// ---- FBs_SlaveControllers/FB_SlaveCtrlMasterSlave.TcPOU
// Brief: Slave Arm MasterSlave controller
FUNCTION_BLOCK PUBLIC FB_SlaveCtrlMasterSlave EXTENDS FB_SlaveArmCtrlBase
VAR_INPUT
END_VAR
VAR_OUTPUT
END_VAR
VAR
	// pose track control kp
	m_posTrackKp :REAL := 0;
	m_oriTrackKp :REAL := 100;
	
	// minimum distance between instrument tip and remote center
	m_minInstruRCDis:LREAL := 0.05;
	
	// master-slave motion scale
	m_MSMotionScale :LREAL;
		
	// gripper match angle threshold
	m_gripperMatchAngThres :LREAL := 2*g_deg2Rad;
	
	// control error thershold from joint limit back to free space
	m_jntLimitOriErr :LREAL :=g_deg2Rad * 5;
	
	// master-slave error thershold to halt control 
	m_safetyOriErr :LREAL :=g_deg2Rad * 150;
	
	// filter cut-off frequency for master-slave control
	m_macroCmdJntPosLpfCutoffFreq : LREAL :=5;
	m_microCmdJntPosLpfCutoffFreq : LREAL :=15;
	
	// last command joint position
	m_lastCmdJntPos :Vec8d;
	
	// simulated DH joint position
	m_simDHJntPos : Vec6d;
	
	// simulated slave twist of DH joint
	m_simDHJointVel :Vec6d;
		
	// enter master-slave control for the first time
	m_firstIn :BOOL := TRUE;
	
	// flag if reach joint limit
	m_reachMacroJntLimit :BOOL;
	m_reachWristJntLimit :BOOL;
	m_jntLimitFlag :Vec6b;
	
	// master/slave origin pose when first enter master-slave control
	m_masterOriginPose : ST_Frame;
	m_slaveOriginPose : ST_Frame;
	
	// orientation deviation(in master coordinate) between master and slave when first enter control
	m_MSOriDeviation : Mat3d;
	
	// command joint position filter
	m_cmdJntPosLpf:ARRAY[1..8] OF FB_LowPassFilter;
	
	// commmand yaw angle and velocity
	m_cmdYawAngle :LREAL;
	m_cmdYawVel :LREAL;
	
	// comand yaw angle and velocity filter
	m_cmdYawAngLpf : FB_LowPassFilter;
	m_cmdYawVelLpf : FB_LowPassFilter;
	
	// master pose/velocity in monitor coordinate
	m_masterPose :ST_Frame;
	m_masterTwist : Vec6d;
	
	// master grip angle
	m_masterGripAngle : LREAL;
	
	// slave command/current pose in endoscope coordinate
	m_slaveCmdPoseInScope :ST_Frame;
	m_slavePoseInScope : ST_Frame;
	
	// slave command/current pose in cart
	m_slaveCmdPoseInCart :ST_Frame;
	m_slavePoseInCart : ST_Frame;
	
	// instrument controller
	m_basicInstruController : FB_BasicInstruControl;
	m_usKnifeController : FB_UltrosonicKnifeControl;
	
	// slave command grip angle and grip force level
	m_slaveCmdGripAngle :LREAL;
	m_slaveCmdGripForceLevel:LREAL;
	
	// slave pose error
	m_slavePosErr :Vec3d;
	m_slaveRotErr :Mat3d;
	m_errAngle : LREAL;
	m_errAxisLocal, m_errAxis :Vec3d;
	m_masterSlavePoseError :Vec6d;
	
	// master velocity in slave coordinate
	m_masterFFVel, m_masterFFWVel :Vec3d;
	
	// velocity for slave to track master motion
	m_slaveCmdVel, m_slaveCmdWVel : Vec3d;
	
	// flag to start gripper control
	m_gripperCtrlFlag :BOOL;
	
	// instrument tyep
	m_instruType : E_InstrumentType;
	
	//################# variable to interpolate master pose ##############
	m_firstInterpolate :BOOL :=TRUE;
	m_lastMasterPose : ST_Frame;
	m_lastMasterGripAngle :LREAL;
	m_masterInterpolateCycle :INT := 4;
	m_curInterpolateCylce :INT := 1;
	m_masterPosInterStep :Vec3d;
	m_masterOriInterStep :Mat3d;
	m_masterGripAngleInterStep :LREAL;
	m_interplotedMasterPose :ST_Frame;
	m_interplotedMasterGripAngle :LREAL;
	
	// code execute time measure
	m_codeTime : Profiler;
	
		m_jnt3Limit :LREAL;
		m_jnt3UB, m_jnt3LB :LREAL;
END_VAR

METHOD PROTECTED calcCmdJntPos : BOOL
VAR_IN_OUT CONSTANT
	i_endoscopePose : ST_Frame;
	i_masterStatus :ST_MasterStatus;
	i_setupStatus: ST_SetupStatus;
	i_slaveArm :FB_SlaveArm;
END_VAR

VAR 
	i,j : INT;
	tmpMat3d : Mat3d;
	masterMotionRange : Vec3d;
	
	masterVelInScope, masterWVelInScope :Vec3d;
	masterVelInCart, masterWVelInCart :Vec3d;

	cmdVelScale :LREAL;
	invJaco :Mat6d;
	armJntJaco,armJntJacoInv, wristJntJaco :Mat3d;
	velByWristJnt,velByArmJnt : Vec3d;
	armDHJntVel, wristDHJntVel :Vec3d;
	tmpFrame : ST_Frame;
	jnt3Limit :LREAL;
	jntDynaUB, jntDynaLB :LREAL;
END_VAR
m_codeTime(START:=TRUE, RESET:=TRUE);

IF isFinished THEN
	RETURN;
END_IF

// decide matched master arm index
FOR i:=1 TO g_mArmNum DO 
	IF i_masterStatus.m_teleSlaveArmIdx[i] = i_slaveArm.armIdx THEN
		masterPoseInterploate(i_masterStatus.m_curArmPose[i],i_masterStatus.m_gripAngle[i]);
		m_masterPose := m_interplotedMasterPose;
		m_masterGripAngle := m_interplotedMasterGripAngle;
		m_masterTwist := i_masterStatus.m_curArmTwist[i];
	END_IF
END_FOR

// compute slave pose in endoscope coordinate
m_slavePoseInCart := transform(i_setupStatus.m_curEndPose[i_slaveArm.armIdx], i_slaveArm.simCartPose);
tmpFrame :=invFrame(i_endoscopePose);
m_slavePoseInScope := transform(tmpFrame, m_slavePoseInCart);

// handle for the first time in
IF TRUE = m_firstIn THEN
	m_firstIn := FALSE;
	m_masterOriginPose :=m_masterPose;
	m_slaveOriginPose := m_slavePoseInScope;
	matTranspose(m_masterOriginPose.m_rot, tmpMat3d);
	matMultiply(tmpMat3d, m_slavePoseInScope.m_rot,m_MSOriDeviation);
	m_lastMasterGripAngle := m_masterGripAngle;
	
	// only update motion scale while entering teleControl 
	m_MSMotionScale := 1.0/ MAX(1,  i_masterStatus.m_motionScale);
END_IF

// compute master twist in slave arm coordinate
FOR i:=1 TO 3 DO
	masterVelInScope[i] := m_masterTwist[i]*m_MSMotionScale;
	masterWVelInScope[i] := m_masterTwist[i+3];
END_FOR
matMultiVec(i_endoScopePose.m_rot, masterVelInScope, masterVelInCart);
matMultiVec(i_endoScopePose.m_rot, masterWVelInScope, masterWVelInCart);
matTranspose(i_setupStatus.m_curEndPose[i_slaveArm.armIdx].m_rot, tmpMat3d);
matMultiVec(tmpMat3d,masterVelInCart, m_masterFFVel);
matMultiVec(tmpMat3d,masterWVelInCart, m_masterFFWVel);

// compute slave command pose in scope
vecSub(m_masterPose.m_pos, m_masterOriginPose.m_pos, masterMotionRange);
vecSelfMultiNum(masterMotionRange, m_MSMotionScale);
vecAdd(m_slaveOriginPose.m_pos, masterMotionRange, m_slaveCmdPoseInScope.m_pos);
matMultiply(m_masterPose.m_rot, m_MSOriDeviation, m_slaveCmdPoseInScope.m_rot);

// compute slave command pose in slave arm coordinate
m_slaveCmdPoseInCart := transform(i_endoScopePose, m_slaveCmdPoseInScope);
tmpFrame := invFrame(i_setupStatus.m_curEndPose[i_slaveArm.armIdx]);
m_cmdCartPose := transform(tmpFrame, m_slaveCmdPoseInCart);

// compute pose error
vecSub(m_cmdCartPose.m_pos, i_slaveArm.simCartPose.m_pos, m_slavePosErr);
matTranspose(i_slaveArm.simCartPose.m_rot, tmpMat3d);
matMultiply(tmpMat3d, m_cmdCartPose.m_rot, m_slaveRotErr);
rot2AngAxis(m_slaveRotErr, angle=>m_errAngle, axis=>m_errAxisLocal);
matMultiVec(i_slaveArm.simCartPose.m_rot, m_errAxisLocal, m_errAxis);

// calculate pose error in endoscope
calcMSErrInScope(i_endoscopePose, i_setupStatus.m_curEndPose[i_slaveArm.armIdx], i_slaveArm);

//safety check
IF ABS(m_errAngle)>m_safetyOriErr THEN
	m_isFinished := TRUE;
	RETURN;
END_IF

// pose track control
vecMultiNum(m_slavePosErr, m_posTrackKp, m_slaveCmdVel);
vecMultiNum(m_errAxis, m_errAngle*m_oriTrackKp, m_slaveCmdWVel);
// final command twist
FOR i:=1 TO 3 DO 
	m_cmdCartTwist[i] := m_slaveCmdVel[i] + m_masterFFVel[i];
	m_cmdCartTwist[i+3] := m_slaveCmdWVel[i] + m_masterFFWVel[i];
END_FOR

// compute command velocity for DH joints
invJaco := i_slaveArm.simJacoInv;
matMultiVec(invJaco, m_cmdCartTwist, m_simDHJointVel);

// limit instrument wrist dofs
limitInstruDofs(i_slaveArm, m_simDHJointVel);

// limit instrument wrist joint velocity
wristLimitSolve(i_slaveArm);

// limit DH joints velocity 
FOR i:=4 TO 6 DO 
	m_simDHJointVel[i] := LIMIT(-GVL_SlaveMotorParameters.g_maxJntVel[i], m_simDHJointVel[i], GVL_SlaveMotorParameters.g_maxJntVel[i]);
END_FOR

// modify arm joints velocity to compensate wrist joint motion
FOR i:=1 TO 3 DO
	FOR j:=1 TO 3 DO
		armJntJaco[i,j]:=i_slaveArm.simJaco[i,j];
		wristJntJaco[i,j]:=i_slaveArm.simJaco[i,j+3];
	END_FOR
	armDHJntVel[i]:=m_simDHJointVel[i];
	wristDHJntVel[i]:=m_simDHJointVel[i+3];
	m_slaveCmdVel[i] := m_cmdCartTwist[i];
END_FOR
invMat3(armJntJaco, armJntJacoInv);
matMultiVec(wristJntJaco, wristDHJntVel, velByWristJnt);
vecSub(m_slaveCmdVel, velByWristJnt, velByArmJnt);
matMultiVec(armJntJacoInv, velByArmJnt, armDHJntVel);

// limit arm joint position
m_reachMacroJntLimit:=false;
FOR i:=1 TO 3 DO
	jntDynaLB := MIN( 0, (GVL_SlaveMotorParameters.g_minDHJntPos[i] - i_slaveArm.simDHJntPos[i])/g_slaveArmCtrlCycleTime);
	IF i=3 THEN
		jnt3Limit := i_slaveArm.instrument.kinematicParameters.m_rodLength+i_slaveArm.instrument.kinematicParameters.m_headLength
											+ i_slaveArm.instrument.kinematicParameters.m_fingerLength - GVL_SlaveArmKinematic.g_minInstruRCDis;
		jntDynaUB := MAX( 0, (jnt3Limit - i_slaveArm.simDHJntPos[i])/g_slaveArmCtrlCycleTime);
		m_jnt3Limit := jnt3Limit;
		m_jnt3UB :=jntDynaUB;
		m_jnt3LB := jntDynaLB;
	ELSE
		jntDynaUB := MAX( 0, (GVL_SlaveMotorParameters.g_maxDHJntPos[i] - i_slaveArm.simDHJntPos[i])/g_slaveArmCtrlCycleTime);
	END_IF
	
	IF m_simDHJointVel[i] >= jntDynaUB OR m_simDHJointVel[i]<= jntDynaLB THEN
		armDHJntVel[i]:=LIMIT(jntDynaLB, m_simDHJointVel[i], jntDynaUB);
		m_reachMacroJntLimit:=TRUE;
	END_IF
END_FOR

// limit DH joints velocity 
FOR i:=1 TO 3 DO
	m_simDHJointVel[i]:=armDHJntVel[i];
	m_simDHJointVel[i+3]:=wristDHJntVel[i];
END_FOR
cmdVelScale := 1;
FOR i:=1 TO g_cartDofs DO 
	cmdVelScale:=MAX(cmdVelScale, ABS(m_simDHJointVel[i]/GVL_SlaveMotorParameters.g_maxJntVel[i]));
END_FOR
vecSelfMultiNum(m_simDHJointVel, 1.0/cmdVelScale);

// integrate command DH joint position
FOR i:=1 TO 6 DO
	m_simDHJntPos[i] := i_slaveArm.simDHJntPos[i] + m_simDHJointVel[i]*g_slaveArmCtrlCycleTime;
END_FOR

// gripper angle/force control
gripperControl(i_slaveArm);

// calculate target motor joint position/velocity from DH joint position
i_slaveArm.instrument.instruIK(m_simDHJntPos,m_slaveCmdGripAngle, o_jntPos=>m_simJntPos);

// filt command joint position
FOR i:=1 TO g_sJntNum DO 
	m_cmdJntPos[i] := m_cmdJntPosLpf[i].run(m_simJntPos[i]);
END_FOR

// compute command joint velocity
vecSub(m_cmdJntPos, m_lastCmdJntPos, m_cmdJntVel);
vecSelfMultiNum(m_cmdJntVel, g_slaveArmCtrlFreq);
m_lastCmdJntPos:=m_cmdJntPos;

m_codeTime(START:=FALSE);
END_METHOD

// override this function in each exact controller
METHOD PROTECTED calcCmdJntTrq : BOOL
VAR_IN_OUT CONSTANT
	i_endoscopePose : ST_Frame;
	i_masterStatus :ST_MasterStatus;
	i_setupStatus: ST_SetupStatus;
	i_slaveArm :FB_SlaveArm;
END_VAR
VAR
	i :INT ;
	instruCmdGripAngle, instruCmdGripForceLevel :LREAL;
	instruCmdJntPos, instruCmdJntVel : Vec5d;	
	instruJntCtrlTrq :Vec5d;
END_VAR
IF isFinished THEN
	RETURN;
END_IF

// set joint torque to zero in default
m_cmdJntTrq := g_zeroVec8d;

// instrument joint control
FOR i:=1 TO 5 DO 
	instruCmdJntPos[i]:=m_cmdJntPos[i+3];
	instruCmdJntVel[i]:=m_cmdJntVel[i+3];
END_FOR
m_cmdYawAngle := m_cmdYawAngLpf.run(m_simDHJntPos[6]);
m_cmdYawVel := m_cmdYawVelLpf.run(m_simDHJointVel[6]);

IF i_slaveArm.instrument.instruType = InstruType_UltrasoundKnifeS OR i_slaveArm.instrument.instruType = InstruType_UltrasoundKnifeU THEN
	m_usKnifeController.run(instruCmdJntPos,instruCmdJntVel, m_slaveCmdGripForceLevel, i_slaveArm, o_cmdJntTrq=>instruJntCtrlTrq);
ELSE
	m_basicInstruController.run(instruCmdJntPos,instruCmdJntVel, m_cmdYawAngle, m_cmdYawVel, m_slaveCmdGripForceLevel, i_slaveArm, o_cmdJntTrq=>instruJntCtrlTrq);
END_IF

FOR i:=1 TO 5 DO
	m_cmdJntTrq[i+3]:=instruJntCtrlTrq[i];
END_FOR
END_METHOD

METHOD calcMSErrInScope : BOOL
VAR_IN_OUT CONSTANT
	i_endoscopePose : ST_Frame;
	i_setupPose :ST_Frame;
	i_slaveArm :FB_SlaveArm;
END_VAR
VAR
	posErrInCart,oriErrInCart :Vec3d;
	invRot :Mat3d;
	posErrInScope,oriErrInScope :Vec3d;
	i:INT;
END_VAR
m_masterSlavePoseError := g_zeroVec6d;

// pose error caused by joints limits
IF m_reachMacroJntLimit OR m_reachWristJntLimit THEN
	// pose error in cart coordinate
	matMultiVec(i_setupPose.m_rot, m_slavePosErr, posErrInCart);
	matMultiVec(i_setupPose.m_rot, m_errAxis, oriErrInCart);
	vecSelfMultiNum(oriErrInCart, m_errAngle);
	
	// pose err in endoscope coordinate
	matTranspose(i_endoscopePose.m_rot, invRot);
	matMultiVec(invRot, posErrInCart, posErrInScope);
	matMultiVec(invRot, oriErrInCart, oriErrInScope);
	
	FOR i:=1 TO 3 DO 
		m_masterSlavePoseError[i]:=posErrInScope[i];
		m_masterSlavePoseError[i+3]:=oriErrInScope[i];
	END_FOR

END_IF
END_METHOD

METHOD gripperControl : BOOL
VAR_IN_OUT CONSTANT
	i_slaveArm :FB_SlaveArm;
END_VAR

VAR
	matchedSlaveGripAngle:LREAL;
	matchedSlaveGripForce:LREAL;
	masterGripVelThres :LREAL := 5.0 *g_deg2Rad;
END_VAR
// compute matched slave grip angle and force
i_slaveArm.instrument.gripAngleMap(m_masterGripAngle,o_instruGripAngle=>matchedSlaveGripAngle, o_instruGripForceLevel=>matchedSlaveGripForce);

IF m_gripperCtrlFlag THEN
	m_slaveCmdGripAngle := matchedSlaveGripAngle;
	m_slaveCmdGripForceLevel := matchedSlaveGripForce;
	RETURN;
ELSE
	//m_gripperCtrlFlag := (ABS(m_masterGripAngleVel) >masterGripVelThres) AND  (m_masterGripAngleVel * (matchedSlaveGripAngle-i_slaveArm.curGripAngle)>0);
	m_gripperCtrlFlag := ABS(matchedSlaveGripAngle-i_slaveArm.curGripAngle)<m_gripperMatchAngThres OR 
	     (matchedSlaveGripAngle>=i_SlaveArm.instrument.kinematicParameters.m_maxGripAngle - m_gripperMatchAngThres AND i_slaveArm.curGripAngle>=matchedSlaveGripAngle) OR 
		(matchedSlaveGripAngle<=i_SlaveArm.instrument.kinematicParameters.m_minGripAngle + m_gripperMatchAngThres AND i_slaveArm.curGripAngle<=matchedSlaveGripAngle);
END_IF
END_METHOD

METHOD PUBLIC init : BOOL
VAR_IN_OUT CONSTANT
	i_slaveArm	:FB_SlaveArm;
END_VAR
VAR_IN_OUT 
	r_slaveArmCtrlCmd :ST_SlaveArmCtrlCmds;
END_VAR
VAR 
	i :INT ;
END_VAR
SUPER^.Init(i_slaveArm,r_slaveArmCtrlCmd);
m_simJntPos :=m_cmdJntPos;
m_lastCmdJntPos :=m_cmdJntPos;
m_jntOPMode[1] := DriverOPMode_PosTrq;
m_jntOPMode[2] := DriverOPMode_PosTrq;
m_jntOPMode[3] := DriverOPMode_PosTrq;
m_jntOPMode[4] := DriverOPMode_Trq;
m_jntOPMode[5] := DriverOPMode_Trq;
m_jntOPMode[6] := DriverOPMode_Trq;
m_jntOPMode[7] := DriverOPMode_Trq;
m_jntOPMode[8] := DriverOPMode_Trq;
m_firstIn :=TRUE;
m_gripperCtrlFlag :=FALSE;

// init gripper angle
m_slaveCmdGripAngle := i_slaveArm.curGripAngle;
m_slaveCmdGripForceLevel:=0;

// init filter
FOR i:=1 TO 3 DO
	m_cmdJntPosLpf[i].init(1, m_macroCmdJntPosLpfCutoffFreq, g_slaveArmCtrlFreq);
END_FOR
FOR i:=4 TO g_sJntNum DO
	m_cmdJntPosLpf[i].init(1, m_microCmdJntPosLpfCutoffFreq, g_slaveArmCtrlFreq);
END_FOR
m_cmdYawAngLpf.init(1, m_microCmdJntPosLpfCutoffFreq, g_slaveArmCtrlFreq);
m_cmdYawVelLpf.init(1, m_microCmdJntPosLpfCutoffFreq, g_slaveArmCtrlFreq);

// init controller
m_basicInstruController.init(i_slaveArm);
m_usKnifeController.init(i_slaveArm);
m_instruType := i_slaveArm.instrument.instruType;

// init interpolation data
m_firstInterpolate :=TRUE;
m_curInterpolateCylce := 1;

// update commands to arm
copyCmds(r_slaveArmCtrlCmd);
END_METHOD

PROPERTY InstruBacklash : Vec5d
GET
IF m_instruType = InstruType_UltrasoundKnifeS OR m_instruType = InstruType_UltrasoundKnifeU THEN
	instruBacklash := g_zeroVec5d;
ELSE
	instruBacklash := m_basicInstruController.m_jntBacklash;
END_IF
END_GET
END_PROPERTY

// limit specific joint dofs based on instrument types
METHOD PRIVATE limitInstruDofs : BOOL
VAR_IN_OUT CONSTANT
	i_slaveArm :FB_SlaveArm;
END_VAR

VAR_IN_OUT
	r_simDHJointVel :Vec6d;
END_VAR
IF i_slaveArm.instrument.instruType = InstruType_UltrasoundKnifeS OR i_slaveArm.instrument.instruType = InstruType_UltrasoundKnifeU THEN
	r_simDHJointVel[5] :=0;
	r_simDHJointVel[6] :=0;
END_IF
END_METHOD

// every some cycles the data from master robots would be miss, so add this interpolation
METHOD masterPoseInterploate : BOOL
VAR_INPUT
	i_masterPose :ST_FRAME;
	i_masterGripAngle :LREAL;
END_VAR

VAR
	rotT :Mat3d;
	rotErr:Mat3d;
	errAngle:LREAL;
	errAxisLocal :Vec3d;
	tmpMat :Mat3d;
END_VAR
IF m_firstInterpolate THEN
	m_firstInterpolate :=FALSE;
	m_lastMasterGripAngle :=i_masterGripAngle;
	m_lastMasterPose := i_masterPose;
	m_masterPosInterStep :=g_zeroVec3d;
	m_masterOriInterStep :=g_eye3d;
	m_masterGripAngleInterStep :=0.0;
	m_interplotedMasterPose := i_masterPose;
	m_interplotedMasterGripAngle := i_masterGripAngle;
END_IF


// update next interpolation
IF m_curInterpolateCylce > m_masterInterpolateCycle THEN
	vecSub(i_masterPose.m_pos, m_lastMasterPose.m_pos, m_masterPosInterStep);
	vecSelfMultiNum( m_masterPosInterStep, 1.0/INT_TO_LREAL(m_masterInterpolateCycle));
	
	matTranspose(m_lastMasterPose.m_rot, rotT);
	matMultiply(rotT, i_masterPose.m_rot, rotErr);
	rot2AngAxis(rotErr, angle=>errAngle, axis=>errAxisLocal);
	m_masterOriInterStep := angAxis2Rot(errAngle/INT_TO_LREAL(m_masterInterpolateCycle), errAxisLocal);
	
	m_masterGripAngleInterStep := (i_masterGripAngle- m_lastMasterGripAngle)/INT_TO_LREAL(m_masterInterpolateCycle);
	
	m_curInterpolateCylce :=1;
	m_lastMasterPose:= i_masterPose;
	m_lastMasterGripAngle := i_masterGripAngle;
END_IF

// control points
IF m_curInterpolateCylce = m_masterInterpolateCycle THEN
	m_interplotedMasterGripAngle := m_lastMasterGripAngle;
	m_interplotedMasterPose := m_lastMasterPose;
// interpolation
ELSE
	m_interplotedMasterGripAngle := m_interplotedMasterGripAngle + m_masterGripAngleInterStep;
	vecSelfAdd(m_interplotedMasterPose.m_pos, m_masterPosInterStep);
	tmpMat := m_interplotedMasterPose.m_rot;
	matMultiply(tmpMat, m_masterOriInterStep, m_interplotedMasterPose.m_rot);
END_IF

m_curInterpolateCylce:= m_curInterpolateCylce+1;
END_METHOD

PROPERTY masterSlavePoseErr : REFERENCE to Vec6d
GET
masterSlavePoseErr REF= m_masterSlavePoseError;
END_GET
END_PROPERTY

// calculate optimized wrist joint velocity when joint limit is violated
METHOD wristLimitSolve : BOOL
VAR_IN_OUT CONSTANT
	i_slaveArm :FB_SlaveArm;
END_VAR

VAR
	i,j:INT;
	jntDynaUB, jntDynaLB :LREAL;
	
	dsrWVel:Vec3d;
	wristJntVel :Vec3d;
	wristJaco:Mat3d;
	
	optJntVel:Vec2d;
	partJaco :Mat32;
	partJacoT :Mat23;
	JtJ,JtJInv :Mat2d;
	partJacoPInv:Mat23;
	
	partJacoPinv2 :Vec3d;
	jacoNorm :LREAL;
	
	wVelLocal,wVelWrd:Vec3d;
	matT:Mat3d;
END_VAR
m_reachWristJntLimit := FALSE;

// desire angular velocity from wrist joint
FOR i:=1 TO 3 DO
	wristJntVel[i] := m_simDHJointVel[i+3];
	FOR j:=1 TO 3 DO
		wristJaco[i,j]:= i_slaveArm.simJaco[i+3, j+3];
	END_FOR 
END_FOR
matMultiVec(wristJaco, wristJntVel, dsrWVel);

// check which joint reaches limit
FOR i:=4 TO 6 DO
	m_jntLimitFlag[i] := FALSE;
	jntDynaUB := MAX( 0, (i_slaveArm.instrument.kinematicParameters.m_wristMaxDHJntPos[i-3] - i_slaveArm.simDHJntPos[i])/g_slaveArmCtrlCycleTime);
	jntDynaLB := MIN( 0, (i_slaveArm.instrument.kinematicParameters.m_wristMinDHJntPos[i-3] - i_slaveArm.simDHJntPos[i])/g_slaveArmCtrlCycleTime);
	IF m_simDHJointVel[i] >= jntDynaUB OR m_simDHJointVel[i]<=jntDynaLB THEN
		m_simDHJointVel[i]:=LIMIT(jntDynaLB, m_simDHJointVel[i], jntDynaUB);
		m_jntLimitFlag[i]:=TRUE;
		m_reachWristJntLimit := TRUE;
	END_IF
END_FOR

// no limit violated
IF NOT( m_jntLimitFlag[4]) AND NOT(m_jntLimitFlag[5]) AND NOT(m_jntLimitFlag[6]) THEN
	RETURN;
END_IF; 

// all joint reach limit
IF m_jntLimitFlag[4] AND m_jntLimitFlag[5] AND m_jntLimitFlag[6] THEN
	RETURN;
END_IF;

// joint 4 reach limit
IF m_jntLimitFlag[4] AND NOT(m_jntLimitFlag[5]) AND NOT(m_jntLimitFlag[6]) THEN
	// colume 2/3
	partJaco[1,1]:= wristJaco[1,2];
	partJaco[2,1]:= wristJaco[2,2];
	partJaco[3,1]:= wristJaco[3,2];
	
	partJaco[1,2]:= wristJaco[1,3];
	partJaco[2,2]:= wristJaco[2,3];
	partJaco[3,2]:= wristJaco[3,3];
	
	// pinv partJaco
	matTranspose(partJaco, partJacoT);
	matMultiply(partJacoT, partJaco, JtJ);
	IF NOT(invMat2(JtJ, JtJInv)) THEN
		m_simDHJointVel[5] :=0;
		m_simDHJointVel[6] := 0;
		RETURN;
	END_IF
	matMultiply(JtJInv, partJacoT, partJacoPinv);
	
	// desire angular velocity exclusive limited joint motion
	dsrWVel[1] := dsrWVel[1] - wristJaco[1,1] * m_simDHJointVel[4];
	dsrWVel[2] := dsrWVel[2] - wristJaco[2,1] * m_simDHJointVel[4];
	dsrWVel[3] := dsrWVel[3] - wristJaco[3,1] * m_simDHJointVel[4];
	
	//NOTE: special handle for roll limit. avoiding joint5/6 motion caused by pitch limit
	matTranspose(i_slaveArm.simCartPose.m_rot, matT);
	matMultiVec(matT, dsrWVel, wVelLocal);
	wVelLocal[3]:=0;
	matMultiVec(i_slaveArm.simCartPose.m_rot, wVelLocal, dsrWVel);
	
	// solve
	matMultiVec(partJacoPinv, dsrWVel, optJntVel);
	m_simDHJointVel[5] :=optJntVel[1];
	m_simDHJointVel[6] := optJntVel[2];
END_IF

// joint 5 reach limit
IF m_jntLimitFlag[5] AND NOT(m_jntLimitFlag[4]) AND NOT(m_jntLimitFlag[6]) THEN
	// colume 1/3
	partJaco[1,1]:= wristJaco[1,1];
	partJaco[2,1]:= wristJaco[2,1];
	partJaco[3,1]:= wristJaco[3,1];
	
	partJaco[1,2]:= wristJaco[1,3];
	partJaco[2,2]:= wristJaco[2,3];
	partJaco[3,2]:= wristJaco[3,3];
	
	// pinv partJaco
	matTranspose(partJaco, partJacoT);
	matMultiply(partJacoT, partJaco, JtJ);
	IF NOT(invMat2(JtJ, JtJInv)) THEN
		m_simDHJointVel[4] :=0;
		m_simDHJointVel[6] := 0;
		RETURN;
	END_IF
	matMultiply(JtJInv, partJacoT, partJacoPinv);
		
	// desire angular velocity exclusive limited joint motion
	dsrWVel[1] := dsrWVel[1] - wristJaco[1,2] * m_simDHJointVel[5];
	dsrWVel[2] := dsrWVel[2] - wristJaco[2,2] * m_simDHJointVel[5];
	dsrWVel[3] := dsrWVel[3] - wristJaco[3,2] * m_simDHJointVel[5];
	
	//NOTE: special handle for pitch limit. avoiding joint4/6 motion caused by pitch limit
	matTranspose(i_slaveArm.simCartPose.m_rot, matT);
	matMultiVec(matT, dsrWVel, wVelLocal);
	wVelLocal[1]:=0;
	matMultiVec(i_slaveArm.simCartPose.m_rot, wVelLocal, dsrWVel);
	
	// solve
	matMultiVec(partJacoPinv, dsrWVel, optJntVel);
	m_simDHJointVel[4] :=optJntVel[1];
	m_simDHJointVel[6] := optJntVel[2];
END_IF

// joint 6 reach limit
IF m_jntLimitFlag[6] AND NOT(m_jntLimitFlag[4]) AND NOT(m_jntLimitFlag[5]) THEN
	// colume 1/2
	partJaco[1,1]:= wristJaco[1,1];
	partJaco[2,1]:= wristJaco[2,1];
	partJaco[3,1]:= wristJaco[3,1];
	
	partJaco[1,2]:= wristJaco[1,2];
	partJaco[2,2]:= wristJaco[2,2];
	partJaco[3,2]:= wristJaco[3,2];
	
	// pinv partJaco
	matTranspose(partJaco, partJacoT);
	matMultiply(partJacoT, partJaco, JtJ);
	IF NOT(invMat2(JtJ, JtJInv)) THEN
		m_simDHJointVel[4] :=0;
		m_simDHJointVel[5] := 0;
		RETURN;
	END_IF
	matMultiply(JtJInv, partJacoT, partJacoPinv);
		
	// desire angular velocity exclusive limited joint motion
	dsrWVel[1] := dsrWVel[1] - wristJaco[1,3] * m_simDHJointVel[6];
	dsrWVel[2] := dsrWVel[2] - wristJaco[2,3] * m_simDHJointVel[6];
	dsrWVel[3] := dsrWVel[3] - wristJaco[3,3] * m_simDHJointVel[6];
	
	// solve
	matMultiVec(partJacoPinv, dsrWVel, optJntVel);
	m_simDHJointVel[4] :=optJntVel[1];
	m_simDHJointVel[5] := optJntVel[2];
END_IF

// joint 4/5 reach limit
IF m_jntLimitFlag[4] AND m_jntLimitFlag[5] AND NOT(m_jntLimitFlag[6]) THEN
	// pinv partJaco of column 3
	partJacoPinv2[1] := wristJaco[1, 3];
	partJacoPinv2[2] := wristJaco[2, 3];
	partJacoPinv2[3] := wristJaco[3, 3];
	jacoNorm := norm(partJacoPinv2);
	vecSelfMultiNum(partJacoPinv2, 1.0/(jacoNorm*jacoNorm));
		
	// desire angular velocity exclusive limited joint motion
	dsrWVel[1] := dsrWVel[1] - wristJaco[1,1] * m_simDHJointVel[4] - wristJaco[1,2] * m_simDHJointVel[5];
	dsrWVel[2] := dsrWVel[2] - wristJaco[2,1] * m_simDHJointVel[4] - wristJaco[2,2] * m_simDHJointVel[5];
	dsrWVel[3] := dsrWVel[3] - wristJaco[3,1] * m_simDHJointVel[4] - wristJaco[3,2] * m_simDHJointVel[5];
	
	// solve
	m_simDHJointVel[6] := vecDot(partJacoPinv2, dsrWVel);
END_IF

// joint 4/6 reach limit
IF m_jntLimitFlag[4] AND m_jntLimitFlag[6] AND NOT(m_jntLimitFlag[5]) THEN
	// pinv partJaco of column 2
	partJacoPinv2[1] := wristJaco[1, 2];
	partJacoPinv2[2] := wristJaco[2, 2];
	partJacoPinv2[3] := wristJaco[3, 2];
	jacoNorm := norm(partJacoPinv2);
	vecSelfMultiNum(partJacoPinv2, 1.0/(jacoNorm*jacoNorm));
		
	// desire angular velocity exclusive limited joint motion
	dsrWVel[1] := dsrWVel[1] - wristJaco[1,1] * m_simDHJointVel[4] - wristJaco[1,3] * m_simDHJointVel[6];
	dsrWVel[2] := dsrWVel[2] - wristJaco[2,1] * m_simDHJointVel[4] - wristJaco[2,3] * m_simDHJointVel[6];
	dsrWVel[3] := dsrWVel[3] - wristJaco[3,1] * m_simDHJointVel[4] - wristJaco[3,3] * m_simDHJointVel[6];
	
	// solve
	m_simDHJointVel[5] := vecDot(partJacoPinv2, dsrWVel);
END_IF

// joint 5/6 reach limit
IF m_jntLimitFlag[5] AND m_jntLimitFlag[6] AND NOT(m_jntLimitFlag[4]) THEN
	// pinv partJaco of column 4
	partJacoPinv2[1] := wristJaco[1, 1];
	partJacoPinv2[2] := wristJaco[2, 1];
	partJacoPinv2[3] := wristJaco[3, 1];
	jacoNorm := norm(partJacoPinv2);
	vecSelfMultiNum(partJacoPinv2, 1.0/(jacoNorm*jacoNorm));
		
	// desire angular velocity exclusive limited joint motion
	dsrWVel[1] := dsrWVel[1] - wristJaco[1,2] * m_simDHJointVel[5] - wristJaco[1,3] * m_simDHJointVel[6];
	dsrWVel[2] := dsrWVel[2] - wristJaco[2,2] * m_simDHJointVel[5] - wristJaco[2,3] * m_simDHJointVel[6];
	dsrWVel[3] := dsrWVel[3] - wristJaco[3,2] * m_simDHJointVel[5] - wristJaco[3,3] * m_simDHJointVel[6];
	
	// solve
	m_simDHJointVel[4] := vecDot(partJacoPinv2, dsrWVel);
END_IF


// check which joint reaches limit
FOR i:=4 TO 6 DO
	jntDynaUB := MAX( 0, (i_slaveArm.instrument.kinematicParameters.m_wristMaxDHJntPos[i-3] - i_slaveArm.simDHJntPos[i])/g_slaveArmCtrlCycleTime);
	jntDynaLB := MIN( 0, (i_slaveArm.instrument.kinematicParameters.m_wristMinDHJntPos[i-3] - i_slaveArm.simDHJntPos[i])/g_slaveArmCtrlCycleTime);
	IF m_simDHJointVel[i] >= jntDynaUB OR m_simDHJointVel[i]<=jntDynaLB THEN
		m_simDHJointVel[i]:=LIMIT(jntDynaLB, m_simDHJointVel[i], jntDynaUB);
		m_jntLimitFlag[i]:=TRUE;
		m_reachWristJntLimit := TRUE;
	END_IF
END_FOR
END_METHOD

END_FUNCTION_BLOCK

// ---- Mains/SafetyCheck.TcPOU
PROGRAM SafetyCheck
VAR
	// slave robot information, including arm status and cartesian data
	m_slaveStatus AT %I* :ST_slaveStatus;
	
	// slave robot joint data
	m_slaveJointData AT %I* :ST_slaveJointData;
	
	// setup robot information
	m_setupStatus AT %I* :ST_SetupStatus;
	
	// setup robot joint data
	m_setupJointsData AT %I* :ST_SetupJointData;
	
	// master robot data, input from master controller box
	m_masterRobotData AT %I* : MSCommu_MasterStatus;
	
	// error check result
	m_safetyCheckData AT %Q* :ST_SafetyData;
	
	// Output cart status
	m_cartStatus AT%I* : ST_CartStatus;
	
	// cart joint data
	m_cartJointsData AT %I* :ST_CartJointData;
	
	//emergency stop and stop botton
	m_stopButton AT %I*: BOOL;
	m_emergencyStopButton AT %I*: BOOL;
	
	//warning tone
	m_warningTone AT %Q*:ARRAY [1..4] OF BOOL;
	
	m_initFlag:bool;
	
	m_SafetyCheck : Fb_SafetyCheck;
	m_checkVariable : ARRAY[1..g_maxNum] OF checkInputVariable;
	m_EtherCATCheck :ARRAY [1..g_maxNum,1..g_maxArmJoint] OF Fb_EtherCATCheck;
	m_errCode :ARRAY [1..3] OF UDINT;
	i , j: INT;
	
	//error robot data record
	m_dataRecord : Fb_dataRecord;
	
	// original position of remote center point when fisrt enter hold state
	m_dsrRcpPos :ARRAY[1..g_sArmNum] OF Vec3d;
	m_rcpPosErrCounts :ARRAY[1..g_sArmNum] OF INT := [4(0)];
	m_rcpPosErr :ARRAY[1..g_sArmNum] OF Vec3d;		// rcp position error
	m_curJntPosLast : ARRAY [1..g_maxArmNum] OF vec13di;  
	m_armErrCodeRefreshLast : ARRAY [1..4] OF UINT;
	
	m_armsRS:ARRAY [1..g_maxArmNum,1..30] OF RS;//复位优先双稳态器
	m_cartRS:ARRAY [1..30] OF RS;//复位优先双稳态器
	m_scopeArmNoReady : BOOL;
	m_joysticksTrigger : BOOL;
	// wait time before robot init  for ethercat to be statble 
	m_safetyCheckInitWaitTime : LREAL:=0;
	
	m_test : DINT;
END_VAR

// reset data
IF FALSE = m_initFlag  THEN
	FOR i:=1  TO g_sArmNum DO 
		m_safetyCheckData.m_slaveErrFlag[i]:=FALSE;
		m_safetyCheckData.m_setupErrFlag[i]:=FALSE;
		m_safetyCheckData.m_cartErrFlag:=FALSE;
	END_FOR
	m_initFlag:=TRUE;
END_IF

armSafetyCheckInputCast();

armSafetyCheckAllowed();

robotPromptMassageCast();

// wait communication to be stable
IF(m_safetyCheckInitWaitTime<g_robotSafetyCheckWaitTime) THEN
	m_safetyCheckInitWaitTime := m_safetyCheckInitWaitTime+g_setupArmCtrlCycleTime;
	RETURN;
END_IF


FOR i:=1  TO g_maxNum DO
	m_SafetyCheck.systemSafetyCheck(i,m_checkVariable,m_cartJointsData,m_setupJointsData,m_slaveJointData);
END_FOR


//error flag to control
readErrFlag();

//Fault code for UI
m_SafetyCheck.errCodeUpdating();

//The fault code is sent to the UI
GVL_interactUI.g_errIdType3:=m_SafetyCheck.o_ErrCode[3];
GVL_interactUI.g_errIdType2:=m_SafetyCheck.o_ErrCode[2];
GVL_interactUI.g_errIdType1:=m_SafetyCheck.o_ErrCode[1];
GVL_interactUI.g_popupErrorArm1 := m_SafetyCheck.m_armErrCodePopup[1];
GVL_interactUI.g_popupErrorArm2 := m_SafetyCheck.m_armErrCodePopup[2];
GVL_interactUI.g_popupErrorArm3 := m_SafetyCheck.m_armErrCodePopup[3];
GVL_interactUI.g_popupErrorArm4 := m_SafetyCheck.m_armErrCodePopup[4];
FOR i:=1  TO g_sArmNum DO
	IF m_SafetyCheck.m_armErrCodeRefresh[i] <> m_armErrCodeRefreshLast[i] THEN
		GVL_interactUI.g_popupRefresh[i] := 1;
	END_IF
	m_armErrCodeRefreshLast[i] := m_SafetyCheck.m_armErrCodeRefresh[i];
END_FOR

//clear fault
IF GVL_interactUI.g_uiFaultReset=1 OR m_masterRobotData.m_uiResetFault = 1 THEN
	m_SafetyCheck.errFlagReset();
	GVL_interactUI.g_uiFaultReset := 0;
END_IF

//robot record information
m_dataRecord.run(m_checkVariable , m_cartStatus , m_cartJointsData , m_setupStatus , m_slaveStatus , m_setupJointsData , m_slaveJointData );

//m_warningTone := warningTone();

METHOD armSafetyCheckAllowed : BOOL
VAR_INPUT
END_VAR
VAR
	i , j : INT; 
END_VAR
FOR i := 1 TO g_maxArmNum DO
	FOR j := 1 TO g_maxArmJoint DO
		IF j > 5 THEN
			//fault code 16#3003 
			m_SafetyCheck.checkPermit[i].m_linkEncErr[j] := m_checkVariable[i].m_slaveDriverInput[j-g_setupJntNum].m_statusWord<>0;
			//fault code 16#3002 
			m_SafetyCheck.checkPermit[i].m_currentIsNotUpdate[j] :=m_checkVariable[i].m_slaveDriverInput[j-g_setupJntNum].m_statusWord<>0 ;
			//fault code 16#2002
			m_SafetyCheck.checkPermit[i].m_armJntFollowErr[j] := m_checkVariable[i].m_slaveDriverInput[j-g_setupJntNum].m_statusWord = DriverStatusWord_OP ;
			//fault code 16#200B
			m_SafetyCheck.checkPermit[i].m_jntCurrentCtrlErr[j] := m_checkVariable[i].m_slaveDriverOutput[j-g_setupJntNum].m_opMode = DriverOPMode_Trq;
		ELSE
			//fault code 16#3003 
			m_SafetyCheck.checkPermit[i].m_linkEncErr[j] := m_checkVariable[i].m_setupDriverInput[j].m_statusWord<>0;
			//fault code 16#3002
			m_SafetyCheck.checkPermit[i].m_currentIsNotUpdate[j] := m_checkVariable[i].m_setupDriverInput[j].m_statusWord<>0 AND j > 2;
			//fault code 16#2002
			m_SafetyCheck.checkPermit[i].m_armJntFollowErr[j] := m_checkVariable[i].m_setupDriverInput[j].m_statusWord = DriverStatusWord_OP AND j > 2;
			//fault code 16#200B
			m_SafetyCheck.checkPermit[i].m_jntCurrentCtrlErr[j] := m_checkVariable[i].m_setupDriverOutput[j].m_opMode = DriverOPMode_Trq AND j > 2;
			
		END_IF
		//fault code 16#3002
		m_SafetyCheck.checkPermit[i].m_jntStatusErr[j] := TRUE;
		//fault code 16#3004
		m_SafetyCheck.checkPermit[i].m_driveErr[j] := TRUE;
		//fault code 16#3005
		m_SafetyCheck.checkPermit[i].m_armJntEncErr[j] := TRUE;
		//fault code 16#3006
		m_SafetyCheck.checkPermit[i].m_outOfLimit[j] := TRUE;
		//fault code 16#3008
		m_SafetyCheck.checkPermit[i].m_motPhieErr[j] := TRUE;
		//fault code 16#2003
		m_SafetyCheck.checkPermit[i].m_jntVelErr[j] := TRUE;
		//fault code 16#2004
		m_SafetyCheck.checkPermit[i].m_spacePoseErr[j] := m_slaveStatus.m_armState[i] = SlaveArmState_MasterSlave AND  norm(m_slaveStatus.m_masterSlavePoseError[i])<g_smallNum;
		//fault code 16#2005
		m_SafetyCheck.checkPermit[i].m_jntCurrentErr[j] := TRUE;
		//fault code 16#2007
		m_SafetyCheck.checkPermit[i].m_fixedPointErr := m_slaveStatus.m_armState[i] = SlaveArmState_MasterSlave;
		//fault code 16#2008
		m_SafetyCheck.checkPermit[i].m_cmdJntSaltation[j] := m_slaveStatus.m_armState[i] = SlaveArmState_MasterSlave;
		//fault code 16#200F
		m_SafetyCheck.checkPermit[i].m_instruOpenAngle := FALSE;
	END_FOR
END_FOR
END_METHOD

METHOD armSafetyCheckInputCast : BOOL
VAR_INPUT
END_VAR

VAR
	i , j: INT; 
END_VAR
FOR i := 1 TO g_maxArmNum DO
	//emergency stop 、stop button and ui stop 
	m_checkVariable[i].EmergencyStop := m_emergencyStopButton;
	m_checkVariable[i].PCStopButton := GVL_interactUI.g_stopButtonFormUI;
	m_checkVariable[i].SlaveStopButton := m_stopButton;
	m_checkVariable[i].MasterStopButton := m_masterRobotData.m_masterStopButton;
	
	IF m_setupStatus.m_armState[i] <> SetupArmState_Hold THEN
		m_dsrRcpPos[i] := m_setupStatus.m_rcPos[i];
	END_IF
	m_checkVariable[i].m_rcpCheck := m_SafetyCheck.rcpErrCheck(m_dsrRcpPos[i],  m_setupStatus.m_rcPos[i], m_rcpPosErrCounts[i] ,m_rcpPosErr[i]);
	m_checkVariable[i].m_spacePoseErr := m_SafetyCheck.poseErrCheck(m_slaveStatus.m_cmdArmPose[i], m_slaveStatus.m_simArmPose[i] );
	
	//slave robot input cast
	FOR j:=1 TO  g_sJntNum DO 		
		m_checkVariable[i].m_slaveDriverInput[j].m_current := SlaveArmControl.m_slaveRobot.m_slaveArms[i].m_joints[j].m_motorInputs.m_current;
		m_checkVariable[i].m_slaveDriverInput[j].m_driverError := SlaveArmControl.m_slaveRobot.m_slaveArms[i].m_joints[j].m_motorInputs.m_driverError;
		m_checkVariable[i].m_slaveDriverInput[j].m_electriAngleDev := SlaveArmControl.m_slaveRobot.m_slaveArms[i].m_joints[j].m_motorInputs.m_electriAngleDev;
		m_checkVariable[i].m_slaveDriverInput[j].m_linkEncoder := SlaveArmControl.m_slaveRobot.m_slaveArms[i].m_joints[j].m_motorInputs.m_linkEncoder;
		m_checkVariable[i].m_slaveDriverInput[j].m_motorEncoder := SlaveArmControl.m_slaveRobot.m_slaveArms[i].m_joints[j].m_motorInputs.m_motorEncoder;
		m_checkVariable[i].m_slaveDriverInput[j].m_statusWord := SlaveArmControl.m_slaveRobot.m_slaveArms[i].m_joints[j].m_motorInputs.m_statusWord;
		IF ABS(m_checkVariable[i].m_slaveDriverInput[j].m_electriAngleDev) > 65536 THEN
			m_test := SlaveArmControl.m_slaveRobot.m_slaveArms[i].m_joints[j].m_motorInputs.m_electriAngleDev;
		END_IF
		//3 joint drive error word at number 6 , move one bit to the right to align with the other joints
		IF j = 3 THEN
			m_checkVariable[i].m_slaveDriverInput[j].m_driverError := SHR(SlaveArmControl.m_slaveRobot.m_slaveArms[i].m_joints[j].m_motorInputs.m_driverError,1);
		END_IF
		m_checkVariable[i].m_slaveDriverOutput[j] := SlaveArmControl.m_slaveRobot.m_slaveArms[i].m_joints[j].m_motorOutputs;
		m_checkVariable[i].m_EtherCATState[j+g_setupJntNum] := m_EtherCATCheck[i,j+g_setupJntNum].EtherCATVerify(GVL_SlaveJointEncoderCaliData.g_slaveArmNetID[i],g_JointNetPort[j+g_setupJntNum]);
		m_checkVariable[i].m_motorEncoderSaltaValue[j+g_setupJntNum] := ABS(m_checkVariable[i].m_slaveDriverInput[j+g_setupJntNum].m_motorEncoder - m_curJntPosLast[i][j+g_setupJntNum]);
		m_curJntPosLast[i][j+g_setupJntNum] := m_checkVariable[i].m_slaveDriverInput[j+g_setupJntNum].m_motorEncoder;
	END_FOR
	
	//setup robot input cast
	FOR j:=1 TO  g_setupJntNum DO 		
		m_checkVariable[i].m_setupDriverInput[j] := SetupArmControl.m_setupRobot.m_setupArms[i].m_joints[j].m_motorInputs;
		m_checkVariable[i].m_setupDriverOutput[j] := SetupArmControl.m_setupRobot.m_setupArms[i].m_joints[j].m_motorOutputs;
		m_checkVariable[i].m_EtherCATState[j] := m_EtherCATCheck[i,j].EtherCATVerify(GVL_SlaveJointEncoderCaliData.g_slaveArmNetID[i],g_JointNetPort[j]);
		m_checkVariable[i].m_motorEncoderSaltaValue[j] := m_checkVariable[i].m_setupDriverInput[j].m_motorEncoder - m_curJntPosLast[i][j];
		m_curJntPosLast[i][j] := m_checkVariable[i].m_setupDriverInput[j].m_motorEncoder;
	END_FOR

END_FOR

//setup robot in-out variable cast
FOR j:=1 TO  g_cartJntNum DO
	m_checkVariable[5].EmergencyStop := m_emergencyStopButton;
	m_checkVariable[5].PCStopButton := GVL_interactUI.g_stopButtonFormUI;
	m_checkVariable[5].SlaveStopButton := m_stopButton;
	m_checkVariable[5].m_cartDriverInput[j] := CartControl.m_cartRobot.m_slaveCart.m_cartJoints[j].m_motorInputs;
	m_checkVariable[5].m_cartDriverOutput[j] := CartControl.m_cartRobot.m_slaveCart.m_cartJoints[j].m_motorOutputs;
	m_checkVariable[5].m_cartEtherCATState[j] := m_EtherCATCheck[5,j].EtherCATVerify(GVL_CartJointEncoderCaliData.g_slaveCartNetID,GVL_CartJointEncoderCaliData.g_slaveCartJointNetPort[j]);
END_FOR
END_METHOD

METHOD joystickAdjust : BOOL
VAR_IN_OUT CONSTANT
	i_joystickValue : vec8d;
END_VAR

VAR
	i : INT;
END_VAR

FOR i := 1 TO 4 DO
	IF 492 > i_joystickValue[i] OR i_joystickValue[i] > 532 THEN
		joystickAdjust := TRUE;
		EXIT;
	END_IF
END_FOR
END_METHOD

METHOD readErrFlag : BOOL
VAR_INPUT
END_VAR
FOR i:=1  TO g_sArmNum DO
	m_safetyCheckData.m_slaveErrFlag[i] := m_SafetyCheck.m_armErrFlag[i,2] OR m_SafetyCheck.m_armErrFlag[i,3];
	m_safetyCheckData.m_setupErrFlag[i] := m_SafetyCheck.m_armErrFlag[i,2] OR m_SafetyCheck.m_armErrFlag[i,3];
END_FOR


GVL_interactUI.g_slaveRecoverErrFlag := BOOL_TO_INT((m_SafetyCheck.m_armErrFlag[1,2] OR m_SafetyCheck.m_armErrFlag[2,2] OR m_SafetyCheck.m_armErrFlag[3,2] OR m_SafetyCheck.m_armErrFlag[4,2]
														OR m_SafetyCheck.m_armErrFlag[g_cartNum,2] OR m_SafetyCheck.m_jntErrFlag[g_cartNum,0,2]) AND GVL_interactUI.g_slaveRunAlone) ;

//cart error flag
m_safetyCheckData.m_cartErrFlag := m_SafetyCheck.m_armErrFlag[g_cartNum,2] OR m_SafetyCheck.m_armErrFlag[g_cartNum,3];
//cart stead foot error flag
m_safetyCheckData.m_cartSteadyFootErr := m_SafetyCheck.m_jntErrFlag[g_cartNum,1,2] OR m_SafetyCheck.m_jntErrFlag[g_cartNum,1,3] 
																	OR m_SafetyCheck.m_jntErrFlag[g_cartNum,2,2] OR m_SafetyCheck.m_jntErrFlag[g_cartNum,2,3] OR m_SafetyCheck.m_jntErrFlag[g_cartNum,0,2];
//cart wheel error flag
m_safetyCheckData.m_cartWheelErr := m_SafetyCheck.m_jntErrFlag[g_cartNum,3,2] OR m_SafetyCheck.m_jntErrFlag[g_cartNum,3,3]
																OR m_SafetyCheck.m_jntErrFlag[g_cartNum,4,2] OR m_SafetyCheck.m_jntErrFlag[g_cartNum,4,3] OR m_SafetyCheck.m_jntErrFlag[g_cartNum,0,2];
//cart stand column error flag
m_safetyCheckData.m_cartStandColumnErr := m_SafetyCheck.m_jntErrFlag[g_cartNum,5,2] OR m_SafetyCheck.m_jntErrFlag[g_cartNum,5,3] OR m_SafetyCheck.m_jntErrFlag[g_cartNum,0,2];
//cart adjust joint contains 6, 7, and 8 joints
m_safetyCheckData.m_cartAdjustErr := m_SafetyCheck.m_jntErrFlag[g_cartNum,6,2] OR m_SafetyCheck.m_jntErrFlag[g_cartNum,6,3] 
															OR m_SafetyCheck.m_jntErrFlag[g_cartNum,7,2] OR m_SafetyCheck.m_jntErrFlag[g_cartNum,7,3]
															OR m_SafetyCheck.m_jntErrFlag[g_cartNum,8,2] OR m_SafetyCheck.m_jntErrFlag[g_cartNum,8,3] OR m_SafetyCheck.m_jntErrFlag[g_cartNum,0,2];
//cart overhang error flag
m_safetyCheckData.m_cartOverhangErr := m_SafetyCheck.m_jntErrFlag[g_cartNum,8,2] OR m_SafetyCheck.m_jntErrFlag[g_cartNum,8,3] OR m_SafetyCheck.m_jntErrFlag[g_cartNum,0,2] OR NOT m_emergencyStopButton;
END_METHOD

METHOD robotPromptMassageCast : BOOL
VAR_IN_OUT CONSTANT
END_VAR

VAR
	i : UDINT;
	m_uiCtrlAdjustFlag : BOOL;
	m_uiCtrlJoystickEnable : BOOL;
	instrument: INT;
END_VAR
FOR i := 1 TO 4 DO
	//0*1021
	m_armsRS[i,1](SET:= m_slaveStatus.m_panelClampErrId[i]=1, 
							RESET1:= NOT m_slaveStatus.m_panelInstallStatus[i], 
							Q1=> m_checkVariable[i].m_promptStatus[1]);
	m_checkVariable[i].m_promptLocation[1] := i + 3;
							
	//0*1022		
	m_armsRS[i,2](SET:= m_slaveStatus.m_panelClampErrId[i]=2, 
							RESET1:= NOT m_slaveStatus.m_panelInstallStatus[i], 
							Q1=> m_checkVariable[i].m_promptStatus[2]);
	m_checkVariable[i].m_promptLocation[2] := i + 3;
	
	//0*1023				
	m_armsRS[i,3](SET:= m_slaveStatus.m_instruReadErrId[i]=1, 
							RESET1:= NOT m_armsRS[i,3].SET OR NOT m_slaveStatus.m_instruInstallStatus[i] , 
							Q1=> m_checkVariable[i].m_promptStatus[3]);
	m_checkVariable[i].m_promptLocation[3] := i + 3;
						
	//0*1024	
	m_armsRS[i,4](SET:= m_slaveStatus.m_instruReadErrId[i]=2, 
							RESET1:=NOT m_armsRS[i,4].SET OR NOT m_slaveStatus.m_instruInstallStatus[i], 
							Q1=> m_checkVariable[i].m_promptStatus[4]);
	m_checkVariable[i].m_promptLocation[4] := i + 3;
	
	//0*1025
	m_armsRS[i,5](SET:= m_slaveStatus.m_instruClampErrId[i]=1, 
							RESET1:=NOT m_armsRS[i,5].SET OR NOT m_slaveStatus.m_instruInstallStatus[i], 
							Q1=> m_checkVariable[i].m_promptStatus[5]);
	m_checkVariable[i].m_promptLocation[5] := i + 3;
	
	 //0*1026
	m_armsRS[i,6](SET:= m_slaveStatus.m_instruClampErrId[i]=2, 
							RESET1:=NOT m_armsRS[i,6].SET OR NOT m_slaveStatus.m_instruInstallStatus[i], 
							Q1=> m_checkVariable[i].m_promptStatus[6]);
	m_checkVariable[i].m_promptLocation[6] := i + 3;
	
	//0*1027
	m_armsRS[i,7](SET:= m_slaveStatus.m_instruReadErrId[i]=3, 
							RESET1:=NOT m_armsRS[i,7].SET OR NOT m_slaveStatus.m_instruInstallStatus[i], 
							Q1=> m_checkVariable[i].m_promptStatus[7]);
	m_checkVariable[i].m_promptLocation[7] := i + 3;
	
	//0*1028	
	m_armsRS[i,8](SET:=NOT m_slaveStatus.m_selfCheckPass[i] AND m_slaveStatus.m_panelInstallStatus[i], 
							RESET1:= NOT m_armsRS[i,8].SET, 
							Q1=> m_checkVariable[i].m_promptStatus[8]);
	m_checkVariable[i].m_promptLocation[8] := i + 3;
				
	//0*1029
	
	 //0*102A
	//m_armsRS[i,10](SET:= m_slaveStatus.m_instruInstallStatus[i] AND NOT m_slaveStatus.m_trocarOnFlag[i], 
	//						RESET1:= NOT m_armsRS[i,10].SET, 
	//						Q1=> m_checkVariable[i].m_promptStatus[10]);
	//m_checkVariable[i].m_promptLocation[10] := i + 3;	
	
	 //0*102B
	FOR j:=1 TO g_mArmNum DO 
		IF i = m_masterRobotData.m_teleSlaveArmIdx[j] THEN
			m_armsRS[i,11](SET:=m_slaveStatus.m_armState[i] = SlaveArmState_Disable AND m_masterRobotData.m_tryMSControl[j] =1, 
									RESET1:= NOT m_armsRS[i,11].SET, 
									Q1=> m_checkVariable[i].m_promptStatus[11]);
			m_checkVariable[i].m_promptLocation[11] := i + 3;
		END_IF
	END_FOR
	
	//0*102C
	FOR j:=1 TO g_mArmNum DO 
		IF i = m_masterRobotData.m_teleSlaveArmIdx[j] THEN
			m_armsRS[i,12](SET:=NOT (SlaveArmState_InstruReady<= m_slaveStatus.m_armState[i] AND m_slaveStatus.m_armState[i] <= SlaveArmState_EndoScope) AND m_masterRobotData.m_tryMSControl[j] =1 AND m_slaveStatus.m_instruStauts[i].m_ready AND m_slaveStatus.m_armState[i] <> SlaveArmState_Disable, 
									RESET1:= NOT m_armsRS[i,12].SET, 
									Q1=> m_checkVariable[i].m_promptStatus[12]);
			m_checkVariable[i].m_promptLocation[12] := i + 3;
		END_IF
	END_FOR
	
				
	//0*102D
	m_armsRS[i,13](SET:= norm(m_slaveStatus.m_masterSlavePoseError[i]) > g_smallNum AND m_slaveStatus.m_armState[i] = SlaveArmState_MasterSlave, 
							RESET1:= NOT m_armsRS[i,13].SET, 
							Q1=> m_checkVariable[i].m_promptStatus[13]);
	m_checkVariable[i].m_promptLocation[13] := i + 3;
	
	
	//0*102E
	m_armsRS[i,14](SET:= NOT SlaveArmControl.m_slaveRobot.m_panelMountedFlag[i] AND (m_masterRobotData.m_tryMSControl[1] =1 OR m_masterRobotData.m_tryMSControl[2] =1) AND m_slaveStatus.m_selfCheckPass[i],
							RESET1:= NOT m_armsRS[i,14].SET, 
							Q1=> m_checkVariable[i].m_promptStatus[14]);
	m_checkVariable[i].m_promptLocation[14] := i + 3;		
	
	//0*102F
	IF InstruType_endoscope = m_slaveStatus.m_instruStauts[i].m_type AND m_slaveStatus.m_endoscopeMounted THEN
		m_scopeArmNoReady := m_slaveStatus.m_armState[i] <> SlaveArmState_ScopeReady AND m_slaveStatus.m_armState[i] <> SlaveArmState_EndoScope;
		m_armsRS[i,15](SET:= (NOT m_slaveStatus.m_endoscopeMounted OR m_scopeArmNoReady) AND (m_masterRobotData.m_tryMSControl[1] =1 OR m_masterRobotData.m_tryMSControl[2] =1), 
								RESET1:= NOT m_armsRS[i,15].SET, 
								Q1=> m_checkVariable[i].m_promptStatus[15]);
		m_checkVariable[i].m_promptLocation[15] := i + 3;	
	ELSE
		m_checkVariable[i].m_promptStatus[15] := FALSE;
	END_IF
END_FOR

//0*102F		预留  没有卡接内窥镜时的检测	
//m_cartRS[15](SET:= NOT m_slaveStatus.m_endoscopeMounted AND (m_masterStatus.m_tryMSControl[1] =1 OR m_masterStatus.m_tryMSControl[2] =1), 
//						RESET1:= NOT m_cartRS[15].SET, 
//						Q1=> m_checkVariable[g_cartNum].m_promptStatus[15]);
//m_checkVariable[g_cartNum].m_promptLocation[15] := 16#0C;


//0*1030			
m_cartRS[16](SET:= NOT m_slaveStatus.m_masterOnLine, 
						RESET1:= m_slaveStatus.m_masterOnLine, 
						Q1=> m_checkVariable[g_cartNum].m_promptStatus[16]);
m_checkVariable[g_cartNum].m_promptLocation[16] := 16#0C;

//0*1031
m_cartRS[17](SET:=m_cartStatus.m_cartDumpEnergy <= 30 , 
						RESET1:= m_cartStatus.m_cartDumpEnergy>30, 
						Q1=> m_checkVariable[g_cartNum].m_promptStatus[17]);
m_checkVariable[g_cartNum].m_promptLocation[17] := g_cartNum + 3;

//0*1032	

//0*1033
m_cartRS[19](SET:= m_cartStatus.m_sdrivingLeverSensorManualFlag, 
						RESET1:=NOT m_cartStatus.m_sdrivingLeverSensorManualFlag, 
						Q1=> m_checkVariable[g_cartNum].m_promptStatus[19]);
m_checkVariable[g_cartNum].m_promptLocation[19] := g_cartNum + 3;

 //0*1034
m_uiCtrlJoystickEnable := m_cartStatus.m_uiControl.m_cameraJoystickEnable OR m_cartStatus.m_uiControl.m_joystickEnable;
m_joysticksTrigger :=  joystickAdjust(m_cartStatus.m_joystickValue);
m_cartRS[20](SET:= m_cartStatus.m_trocarOnFlag=0 AND NOT m_uiCtrlJoystickEnable AND m_joysticksTrigger, 
						RESET1:= NOT m_cartRS[20].SET, 
						Q1=> m_checkVariable[g_cartNum].m_promptStatus[20]);
m_checkVariable[g_cartNum].m_promptLocation[20] := g_cartNum + 3;
					
//0*1035
m_uiCtrlAdjustFlag := m_cartStatus.m_uiControl.m_cameraJoystickEnable OR m_cartStatus.m_uiControl.m_dockingEnable OR m_cartStatus.m_uiControl.m_drapingEnable
							OR m_cartStatus.m_uiControl.m_joystickEnable OR m_cartStatus.m_uiControl.m_packageEnable;
m_cartRS[21](SET:= m_cartStatus.m_trocarOnFlag>0 AND m_uiCtrlAdjustFlag, 
						RESET1:= m_cartStatus.m_trocarOnFlag=0 OR NOT m_uiCtrlAdjustFlag, 
						Q1=> m_checkVariable[g_cartNum].m_promptStatus[21]);
m_checkVariable[g_cartNum].m_promptLocation[21] := g_cartNum + 3;

//0*1036
m_cartRS[22](SET:= m_cartStatus.m_uiControl.m_joystickEnable AND (m_cartStatus.m_jntPosReachLimit[5] OR m_cartStatus.m_jntPosReachLimit[6] OR m_cartStatus.m_jntPosReachLimit[7] OR m_cartStatus.m_jntPosReachLimit[8]), 
						RESET1:= NOT m_cartRS[22].SET, 
						Q1=> m_checkVariable[g_cartNum].m_promptStatus[22]);
m_checkVariable[g_cartNum].m_promptLocation[22] := g_cartNum + 3;
END_METHOD

METHOD warningTone : vec4b
VAR_INPUT
END_VAR
IF (GVL_interactUI.g_curErrType=3) THEN
	warningTone[1] := TRUE;
	warningTone[2] := FALSE;
	warningTone[3] := FALSE;
ELSIF (GVL_interactUI.g_curErrType=2) THEN
	warningTone[1] := FALSE;
	warningTone[2] := TRUE;
	warningTone[3] := FALSE;
//ELSIF (GVL_interactUI.g_curErrType=1) THEN
//	warningTone[1] := TRUE;
//	warningTone[2] := TRUE;
//	warningTone[3] := FALSE;
ELSIF (CartControl.m_cartRobot.m_slaveCart.m_columnJntVel <> 0 AND NOT CartControl.m_cartRobot.m_slaveCart.m_columnAdjustEnable) THEN
	warningTone[1] := FALSE;
	warningTone[2] := FALSE;
	warningTone[3] := TRUE;
//ELSIF m_cartStatus.m_CartState >= CartJointState_HangAdjust AND  m_cartStatus.m_CartState <= CartJointState_StandColuAdjust THEN
//	warningTone[1] := TRUE;
//	warningTone[2] := FALSE;
//	warningTone[3] := TRUE;
ELSE
	warningTone[1] := FALSE;
	warningTone[2] := FALSE;
	warningTone[3] := FALSE;
END_IF
END_METHOD

END_PROGRAM

// ---- SafetyCheck/Fb_SafetyCheck.TcPOU
FUNCTION_BLOCK Fb_SafetyCheck
VAR_INPUT
END_VAR
VAR_OUTPUT
END_VAR
VAR
	i, j:INT;
	m_checkDelay :ARRAY[1..g_maxNum] OF checkDelay;
	m_checkDelayTime :checkDelayTime;
	m_checkPermit:ARRAY[1..g_maxNum] OF  checkPermit;
	
	m_jntErrFlag:ARRAY[1..g_maxNum,0..g_maxArmJoint,1..3] OF BOOL;
	m_armErrFlag:ARRAY [1..g_maxNum,1..3] OF BOOL;
	m_errCode:UDINT;
	
	
	m_errNumType: ARRAY [1..3] OF INT;
	m_ArrayErrCodeType:ARRAY [1..3] OF ARRAY [0..30] OF UDINT;
	m_ArrayErrCodeTypeTest:ARRAY [1..3] OF ARRAY [0..100] OF UDINT;
	m_armErrCodePopup : ARRAY [1..4] OF ARRAY [0..2] OF UDINT;
	m_armErrCodeRefresh : ARRAY [1..4] OF UINT;
	
	//The fault is sent to the UI at the frequency of 0.1S
	m_errCodeUpdateFlag: ARRAY [1..3] OF BOOL;
	m_errCodeUpdateTon: ARRAY [1..3] OF TON;
	
	m_curJntTorqueIOlast :ARRAY [1..g_maxArmNum] OF vec13di;  
	m_cmdJntPosLast : ARRAY [1..g_maxArmNum] OF vec13d;  
	m_cartCurJntTorqueIOlast :vec8di;  
	m_cartCmdJntPosLast : vec8d;  
	o_ErrCode:ARRAY [1..3] OF UDINT;
		
	m_PromptMassBusy:BOOL;
	m_PromptFlag:ARRAY[1..g_maxNum,1..30] OF UINT;
	m_deleteCode:UDINT;
	
END_VAR


VAR CONSTANT
	m_codeUpdateDelay:TIME:=T#0.1S;
	
	//Fault level: 1 indicates  prompt message, 2 indicates a recoverable fault and 3 indicates an unrecoverable fault
	m_promptMessageLevel : UINT :=1;
	m_rcvLevel : UINT:=2;
	m_unrcvLevel : UINT :=3;
END_VAR

METHOD arrayDeleteFrist : ARRAY [0..30] OF UDINT;
VAR_INPUT
	i_array:ARRAY [0..30] OF UDINT;
END_VAR

VAR
	k:INT;
END_VAR

arrayDeleteFrist[30]:=0;

FOR k:=0 TO 29 BY 1 DO
	arrayDeleteFrist[k]:=i_array[k+1];
END_FOR
END_METHOD

METHOD arrayFILO : ARRAY [0..100] OF  UDINT
VAR_INPUT
	i_array:ARRAY[0..100] OF UDINT;
	i_newData:UDINT;
END_VAR

VAR
	i:INT;
END_VAR

FOR i:=0 TO 20 BY 1 DO
	arrayFILO[i]:=i_array[i];
	IF i_array[i]=0 THEN
		arrayFILO[i]:=i_newData;
		EXIT;
	END_IF
END_FOR
END_METHOD

METHOD cartSafetyCheck : BOOL
VAR_INPUT
	i_armId:UDINT;
	i_safetyCheckVar : checkInputVariable;
	i_cartJointData : ST_CartJointData;
END_VAR


VAR
	k:INT;
END_VAR


//驱动器状态监测、驱动器未连接
FOR i:=1 TO g_maxCartJoint BY 1 DO
	m_checkDelay[i_ArmId].T_cartJntStatusErr[i](IN:= (i_safetyCheckVar.m_cartDriverInput[i].m_statusWord=0 AND m_checkPermit[i_ArmId].m_cartJntStatus[i]), PT:=m_checkDelayTime.Ti_CarJntStatus , Q=> , ET=> );
	IF m_checkDelay[i_ArmId].T_cartJntStatusErr[i].Q THEN
		errCodeAssign(i_ArmId, i_ArmId+3,  0, i, 16#3002 ,m_unrcvLevel );
	END_IF
END_FOR



//关节编码器监测
FOR i:=1 TO g_maxCartJoint BY 1 DO
	m_checkDelay[i_ArmId].T_cartLinkEncErr[i](IN:= (i_safetyCheckVar.m_cartDriverInput[i].m_linkEncoder=g_cartMaxLinkEnc[i] OR i_safetyCheckVar.m_cartDriverInput[i].m_linkEncoder=g_cartMinLinkEnc[i]) AND m_checkPermit[i_ArmId].m_cartJntEncErr[i], PT:=m_checkDelayTime.Ti_CarActSec , Q=> , ET=> );
	IF m_checkDelay[i_ArmId].T_cartLinkEncErr[i].Q THEN
		errCodeAssign(i_ArmId, i_ArmId+3,  0, i, 16#3003 ,m_unrcvLevel );
	END_IF
END_FOR


//驱动器错误检测
FOR i:=1 TO g_maxCartJoint BY 1 DO
	m_checkDelay[i_ArmId].T_cartDriveErr[i](IN:= (i_safetyCheckVar.m_cartDriverInput[i].m_driverError AND 16#20)=32 AND m_checkPermit[i_ArmId].m_cartDriveErr[i] , PT:=m_checkDelayTime.Ti_CarDriveErr , Q=> , ET=> );
	IF m_checkDelay[i_ArmId].T_cartDriveErr[i].Q THEN
		errCodeAssign(i_ArmId, i_ArmId+3,  0, i, 16#3004 ,m_unrcvLevel );
	END_IF
END_FOR



//台车双编码器偏差过大
FOR i:=1 TO g_maxCartJoint BY 1 DO
	m_checkDelay[i_ArmId].T_cartJntEncErr[i](IN:= ABS (i_cartJointData.m_curLinkPos[i]-i_cartJointData.m_curJntPos[i])>g_cartMaxJntEncErr[i] AND m_checkPermit[i_ArmId].m_cartJntEncErr[i], PT:=m_checkDelayTime.Ti_CarDualEncDev , Q=> , ET=> );
	IF m_checkDelay[i_ArmId].T_cartJntEncErr[i].Q THEN
		errCodeAssign(i_ArmId, i_ArmId+3,  0, i, 16#3005 ,m_unrcvLevel );
	END_IF
END_FOR


//关节运动超限位
FOR i:=1 TO g_maxCartJoint BY 1 DO
	m_checkDelay[i_ArmId].T_cartOutOfLimit[i](IN:= (i_cartJointData.m_curJntPos[i]>=g_cartMaxJntPos[i] OR i_cartJointData.m_curJntPos[i]<=g_cartMinJntPos[i]) AND m_checkPermit[i_ArmId].m_cartOutOfLimit[i] , PT:=m_checkDelayTime.Ti_CaroutofLimit , Q=> , ET=> );
	IF m_checkDelay[i_ArmId].T_cartOutOfLimit[i].Q THEN
		errCodeAssign(i_ArmId, i_ArmId+3,  0, i, 16#3006 ,m_unrcvLevel );
	END_IF
END_FOR


//驱动器内部通讯错误
FOR i:=1 TO g_maxCartJoint BY 1 DO
	m_checkDelay[i_ArmId].T_cartCurrentIsNotUpdate[i](IN:= (i_safetyCheckVar.m_cartDriverInput[i].m_current=m_cartCurJntTorqueIOlast[i] AND m_checkPermit[i_ArmId].m_cartCurrentIsNotUpdate[i]), PT:=m_checkDelayTime.Ti_CarTorMotor , Q=> , ET=> );
	IF m_checkDelay[i_ArmId].T_cartCurrentIsNotUpdate[i].Q THEN
		errCodeAssign(i_ArmId, i_ArmId+3,  0, i, 16#3009 ,m_unrcvLevel );
	END_IF
	m_cartCurJntTorqueIOlast[i]:=i_safetyCheckVar.m_cartDriverInput[i].m_current;
END_FOR


//关节跟随误差过大
FOR i:=1 TO g_maxCartJoint BY 1 DO
	m_checkDelay[i_ArmId].T_cartJntFollowErr[i](IN:= ABS(i_cartJointData.m_cmdJntPos[i]- i_cartJointData.m_curJntPos[i])>g_cartMaxJntFollowErr[i]  AND m_checkPermit[i_ArmId].m_cartFollowErr[i], PT:=m_checkDelayTime.Ti_CarFollowDev , Q=> , ET=> );
	IF m_checkDelay[i_ArmId].T_cartJntFollowErr[i].Q THEN
		errCodeAssign(i_ArmId, i_ArmId+3,  0, i, 16#2002 ,m_rcvLevel );
	END_IF
END_FOR


//关节速度监控
FOR i:=1 TO g_maxCartJoint BY 1 DO
	m_checkDelay[i_ArmId].T_cartJntVelErr[i](IN:= ABS(i_cartJointData.m_curJntVel[i])>g_cartMaxJntVel[i] AND m_checkPermit[i_ArmId].m_cartJntVelErr[i], PT:=m_checkDelayTime.Ti_CarJntVel , Q=> , ET=> );
	IF m_checkDelay[i_ArmId].T_cartJntVelErr[i].Q THEN
		errCodeAssign(i_ArmId, i_ArmId+3,  0, i, 16#2003 ,m_rcvLevel );
	END_IF
END_FOR


//电流超限监测
FOR i:=1 TO g_maxCartJoint BY 1 DO
	m_checkDelay[i_ArmId].T_cartJntCurrentErr[i](IN:= ABS(i_cartJointData.m_curJntTrq[i])>g_cartMaxJntCurrent[i] AND m_checkPermit[i_ArmId].m_cartJntCurrentErr[i], PT:=m_checkDelayTime.Ti_CarJntCurrent , Q=> , ET=> );
	IF m_checkDelay[i_ArmId].T_cartJntCurrentErr[i].Q THEN
		errCodeAssign(i_ArmId, i_ArmId+3,  0, i, 16#2005 ,m_rcvLevel );
	END_IF
END_FOR


//Ethercat通讯检测
FOR i:=1 TO g_maxCartJoint BY 1 DO
	IF NOT i_safetyCheckVar.m_cartEtherCATState[i].EtherCATState THEN
		errCodeAssign(i_ArmId, i_ArmId+3,  0, i, 16#2006 ,m_rcvLevel );
	END_IF
END_FOR


//鸣志驱动器错误检测
FOR i:=1 TO g_maxCartJoint BY 1 DO
	m_checkDelay[i_ArmId].T_CarMingzhiDriveErr[i](IN:= (i_safetyCheckVar.m_cartDriverInput[i].m_statusWord AND 16#0F)=15  AND m_checkPermit[i_ArmId].m_cartMZDriveErr[i] , PT:=m_checkDelayTime.Ti_CarMZDriveErr , Q=> , ET=> );
	IF m_checkDelay[i_ArmId].T_CarMingzhiDriveErr[i].Q THEN
		errCodeAssign(i_ArmId, i_ArmId+3,  0, i, 16#2009 ,m_rcvLevel );
	END_IF
END_FOR
END_METHOD

PROPERTY checkPermit : REFERENCE TO ARRAY[1..g_maxNum] OF  checkPermit
GET
checkPermit ref= m_checkPermit;
END_GET
SET
END_SET
END_PROPERTY

METHOD electriAngleDev : DINT
VAR_INPUT
	i_motorElectriAngleDev : DINT;
END_VAR

IF i_motorElectriAngleDev > 50000 THEN
	electriAngleDev := i_motorElectriAngleDev - 65535;
ELSIF i_motorElectriAngleDev < -50000 THEN
	electriAngleDev := i_motorElectriAngleDev + 65535;
ELSE
	electriAngleDev := i_motorElectriAngleDev;
END_IF
END_METHOD

METHOD errCodeAssign : BOOL
VAR_INPUT
	i_armId:UDINT;
	i_errLocation:UDINT;
	i_errCodeMode:UDINT;
	i_errJoint:UDINT;
	i_errID:UDINT;
	i_errFlagID :UINT;
END_VAR
IF m_jntErrFlag[i_armId,i_errJoint,i_errFlagID]=FALSE THEN
	m_jntErrFlag[i_armId,i_errJoint,i_errFlagID]:=TRUE;
	m_errCode:=SHL(i_errLocation,24)+SHL(i_errCodeMode,20)+SHL(i_errJoint,16)+i_errID;
	
	
	IF i_errID>=16#3000 THEN
		m_errNumType[m_unrcvLevel]:=LIMIT(0,m_errNumType[m_unrcvLevel]+1,100);
		m_arrayErrCodeType[m_unrcvLevel][m_errNumType[m_unrcvLevel]]:=m_errCode;
		g_arrayErrCodeArm[i_armId]:=arrayFILO(i_Array:= g_arrayErrCodeArm[i_ArmId], i_NewData:=m_errCode );
		m_armErrFlag[i_armId,m_unrcvLevel]:=TRUE;
		
	ELSIF i_errID>=16#2000 THEN
		m_errNumType[m_rcvLevel]:=LIMIT(0,m_errNumType[m_rcvLevel]+1,100);
		m_arrayErrCodeType[m_rcvLevel][m_errNumType[m_rcvLevel]]:=m_errCode;
		g_arrayErrCodeArm[i_armId]:=arrayFILO(i_Array:= g_arrayErrCodeArm[i_ArmId], i_NewData:=m_errCode );
		m_armErrFlag[i_armId,m_rcvLevel]:=TRUE;
		
	END_IF
END_IF
END_METHOD

METHOD errCodeUpdating :ARRAY [1..3] OF UDINT;
VAR_INPUT
END_VAR

m_errCodeUpdateTon[m_unrcvLevel](IN:= NOT m_errCodeUpdateFlag[3], PT:=m_codeUpdateDelay , Q=> m_errCodeUpdateFlag[3], ET=> );
IF m_errCodeUpdateFlag[m_unrcvLevel] THEN
	IF m_errNumType[m_unrcvLevel]>=1 THEN
		m_ArrayErrCodeType[m_unrcvLevel]:=ArrayDeleteFrist(i_Array:=m_ArrayErrCodeType[3]) ;
		o_ErrCode[m_unrcvLevel]:=m_ArrayErrCodeType[m_unrcvLevel][0] ;
		m_ArrayErrCodeTypeTest[m_unrcvLevel]:=arrayFILO(i_Array:= m_ArrayErrCodeTypeTest[m_unrcvLevel], i_NewData:=o_ErrCode[m_unrcvLevel] );
		m_errNumType[m_unrcvLevel]:=m_errNumType[m_unrcvLevel]-1;
	END_IF
END_IF


m_errCodeUpdateTon[m_rcvLevel](IN:= NOT m_errCodeUpdateFlag[m_rcvLevel], PT:=m_codeUpdateDelay , Q=> m_errCodeUpdateFlag[2], ET=> );
IF m_errCodeUpdateFlag[m_rcvLevel] THEN
	IF m_errNumType[m_rcvLevel]>=1 THEN
		m_ArrayErrCodeType[m_rcvLevel]:=ArrayDeleteFrist(i_Array:=m_ArrayErrCodeType[2]) ;
		o_ErrCode[m_rcvLevel]:=m_ArrayErrCodeType[m_rcvLevel][0] ;
		m_ArrayErrCodeTypeTest[m_rcvLevel]:=arrayFILO(i_Array:= m_ArrayErrCodeTypeTest[m_rcvLevel], i_NewData:=o_ErrCode[m_rcvLevel] );
		m_errNumType[m_rcvLevel]:=m_errNumType[m_rcvLevel]-1;
	END_IF
END_IF
END_METHOD

METHOD errFlagReset : BOOL
VAR_INPUT
END_VAR

FOR i := 1 TO g_maxNum DO
	FOR j :=0 TO g_maxArmJoint DO
		m_jntErrFlag[i, j, 2]:=FALSE;
	END_FOR
	m_armErrFlag[i, 2]:=FALSE;
END_FOR

o_ErrCode[2]:=0;
END_METHOD

METHOD poseErrCheck : vec6d
VAR_INPUT
	i_cmdPose : ST_Frame;
	i_curPose :ST_Frame;
END_VAR

VAR
	posErr,oriErr:Vec3d;
	matT,rotErr:Mat3d;
	errAngle :LREAL;
	errAxis :Vec3d;
	i : INT;
END_VAR
vecSub(i_cmdPose.m_pos, i_curPose.m_pos,posErr);

matTranspose(i_cmdPose.m_rot, matT);
matMultiply(matT,i_curPose.m_rot, rotErr);
rot2AngAxis(rotErr, angle=>errAngle, axis=>errAxis);
vecMultiNum(errAxis, errAngle,oriErr);

FOR i := 1 TO 6 DO
	IF i <= 3 THEN
		poseErrCheck[i] := posErr[i];
	ELSE
		poseErrCheck[i] := oriErr[i];
	END_IF
END_FOR
END_METHOD

METHOD promptMassCode : BOOL
VAR_INPUT
	i_PromptStatus:BOOL;
	i_ArmId:UDINT;
	i_ErrID:UDINT;
	i_ErrLocation:UDINT;
END_VAR
VAR
	m_errStatus : UDINT := 0;
	//error ID , 0-15 bit
	m_errId : UDINT;
	m_arrayErrCode : ARRAY [0..30] OF UDINT;
	m_armErrCode : ARRAY [0..2] OF UDINT;
END_VAR

m_PromptMassBusy:=TRUE;

//prompt flag set true
IF i_PromptStatus=TRUE AND m_PromptFlag[i_ArmId,i_ErrID]=0 THEN
	m_PromptFlag[i_ArmId,i_ErrID]:=1;
END_IF

//
IF i_ErrLocation <= 7 AND i_ErrLocation >= 4 THEN
	m_errStatus := 16#00FF;
ELSE
	m_errStatus := 0;
END_IF
m_errId := i_errID+16#1020;

//output prompt error code
IF m_PromptFlag[i_ArmId,i_ErrID]=1 THEN
	m_ErrCode:=SHL(i_ErrLocation,24)+SHL(m_errStatus,16)+i_errID+16#1020;
	vecFIFO(m_ArrayErrCodeType[1] , m_ErrCode , m_arrayErrCode );
	m_ArrayErrCodeType[1]:=m_arrayErrCode;
	IF (m_ErrCode AND 16#00FF0000) = 16#00FF0000 THEN
		vecFIFO(m_armErrCodePopup[i_armId] , m_ErrCode , m_armErrCode );
		m_armErrCodePopup[i_armId] := m_armErrCode;
		m_armErrCodeRefresh[i_armId] := 1;
	END_IF
	m_PromptFlag[i_ArmId,i_ErrID]:=2;
END_IF

//clear prompt error code
IF m_PromptFlag[i_ArmId,i_ErrID]=2 AND i_PromptStatus=FALSE THEN
	m_deleteCode:=SHL(i_ErrLocation,24)+SHL(m_errStatus,16)+i_ErrID+16#1020;
	vecDeleteInput(m_ArrayErrCodeType[1] , m_deleteCode , m_arrayErrCode);
	m_ArrayErrCodeType[1] := m_arrayErrCode;
	IF (m_deleteCode AND 16#00FF0000)  = 16#00FF0000 THEN
		vecDeleteInput(m_armErrCodePopup[i_armId] , m_deleteCode , m_armErrCode );
		m_armErrCodePopup[i_armId] := m_armErrCode;
		m_armErrCodeRefresh[i_armId] := 2;
	END_IF
	//ArrayDeleteInput(i_Array:= m_ArrayErrCodeType[1], i_DeleteCode:=m_deleteCode , o_Array=> m_ArrayErrCodeType[1]);
	m_PromptFlag[i_ArmId,i_ErrID]:=0;
END_IF
o_ErrCode[1]:=m_ArrayErrCodeType[1][0];
m_PromptMassBusy:=FALSE;
END_METHOD

METHOD rcpErrCheck : BOOL
VAR_INPUT
	i_cmdPos : Vec3d;
	i_curPos : Vec3d;
END_VAR
VAR_IN_OUT
	r_errCount:INT;
	r_posErr :Vec3d;
END_VAR

VAR
	err:Vec3d;
END_VAR
vecSub(i_cmdPos, i_curPos,err);
r_posErr:=err;

IF  (norm(err)>g_rcpDeviationThres) THEN
	r_errCount:= r_errCount +1;
ELSE 
	r_errCount:=0;
END_IF
rcpErrCheck := r_errCount >= g_faultTriggerCounts;
END_METHOD

METHOD setupSafetyCheck : BOOL
VAR_INPUT
	i_armId:UDINT;
	i_safetyCheckVar :ARRAY[1..g_maxNum] OF checkInputVariable;
	i_setupJointData : ST_SetupJointData;
END_VAR

VAR
	k:INT;
END_VAR


//驱动器状态监测、驱动器未连接
FOR i:=1 TO g_setupJntNum BY 1 DO
	m_checkDelay[i_ArmId].T_jntStatusErr[i](IN:= (i_safetyCheckVar[i_ArmId].m_setupDriverInput[i].m_statusWord=0 AND m_checkPermit[i_ArmId].m_jntStatusErr[i]), PT:=m_checkDelayTime.Ti_jntStatusErr , Q=> , ET=> );
	IF m_checkDelay[i_ArmId].T_jntStatusErr[i].Q THEN
		errCodeAssign(i_ArmId, i_ArmId+3,  0, i, 16#3002 ,m_unrcvLevel );
	END_IF
END_FOR



//关节编码器监测
FOR i:=1 TO g_setupJntNum BY 1 DO
	m_checkDelay[i_ArmId].T_linkEncErr[i](IN:= (i_safetyCheckVar[i_ArmId].m_setupDriverInput[i].m_linkEncoder=g_maxLinkEnc[i] OR i_safetyCheckVar[i_ArmId].m_setupDriverInput[i].m_linkEncoder=g_minLinkEnc[i]) AND m_checkPermit[i_ArmId].m_linkEncErr[i], PT:=m_checkDelayTime.Ti_linkEncErr , Q=> , ET=> );
	IF m_checkDelay[i_ArmId].T_linkEncErr[i].Q THEN
		errCodeAssign(i_ArmId, i_ArmId+3,  0, i,  16#3003 ,m_unrcvLevel );
	END_IF
END_FOR


//驱动器错误检测
FOR i:=1 TO g_setupJntNum BY 1 DO
	m_checkDelay[i_ArmId].T_DriveErr[i](IN:= (i_safetyCheckVar[i_ArmId].m_setupDriverInput[i].m_driverError AND 16#20)=g_driveErrWord AND m_checkPermit[i_ArmId].m_driveErr[i] , PT:=m_checkDelayTime.Ti_driveErr , Q=> , ET=> );
	IF m_checkDelay[i_ArmId].T_DriveErr[i].Q THEN
		errCodeAssign(i_ArmId, i_ArmId+3,  0, i, 16#3004 ,m_unrcvLevel );
	END_IF
END_FOR


//双编码器偏差过大检测
FOR i:=1 TO g_setupJntNum BY 1 DO
	m_checkDelay[i_ArmId].T_armJntEncErr[i](IN:= ABS(i_setupJointData.m_curLinkPos[i_armId][i]-i_setupJointData.m_curJntPos[i_armId][i])>=g_armMaxJntEncErr[i] AND m_checkPermit[i_ArmId].m_armJntEncErr[i], PT:=m_checkDelayTime.Ti_armJntEncErr , Q=> , ET=> );
	IF m_checkDelay[i_ArmId].T_armJntEncErr[i].Q THEN
		errCodeAssign( i_ArmId, i_ArmId+3,  0, i, 16#3005, m_unrcvLevel );
	END_IF
END_FOR


//关节运动超限位
FOR i:=1 TO g_setupJntNum BY 1 DO
	m_checkDelay[i_ArmId].T_outOfLimit[i](IN:= (i_setupJointData.m_curJntPos[i_armId][i]>=(g_maxJntPos[i_armId,i]+g_armJntPosLimitBuffer[i]) OR i_setupJointData.m_curJntPos[i_armId][i]<=(g_minJntPos[i_armId,i]-g_armJntPosLimitBuffer[i])) AND m_checkPermit[i_ArmId].m_outOfLimit[i] , PT:=m_checkDelayTime.Ti_outofLimit , Q=> , ET=> );
	IF m_checkDelay[i_ArmId].T_outOfLimit[i].Q THEN
		errCodeAssign(i_ArmId, i_ArmId+3,  0, i, 16#3006, m_unrcvLevel );
	END_IF
END_FOR


//电机电角度偏差
FOR i:=1 TO g_setupJntNum BY 1 DO
	IF ABS(electriAngleDev(i_safetyCheckVar[i_armId].m_setupDriverInput[i].m_electriAngleDev))> g_motPhieErrLimit  AND m_checkPermit[i_ArmId].m_motPhieErr[i] THEN
		errCodeAssign(i_ArmId, i_ArmId+3,  0, i, 16#3008, m_unrcvLevel );
	END_IF
END_FOR


//驱动器内部通讯错误
FOR i:=1 TO g_setupJntNum BY 1 DO
	m_checkDelay[i_ArmId].T_currentIsNotUpdate[i](IN:= (i_safetyCheckVar[i_ArmId].m_setupDriverInput[i].m_current=m_curJntTorqueIOlast[i_ArmId][i] AND m_checkPermit[i_ArmId].m_currentIsNotUpdate[i]), PT:=m_checkDelayTime.Ti_currentIsNotUpdate , Q=> , ET=> );
	IF  m_checkDelay[i_ArmId].T_currentIsNotUpdate[i].Q THEN
		errCodeAssign(i_ArmId, i_ArmId+3,  0, i, 16#3009 ,m_unrcvLevel );
	END_IF
	m_curJntTorqueIOlast[i_ArmId][i]:=i_safetyCheckVar[i_ArmId].m_setupDriverInput[i].m_current;
END_FOR


//关节跟随误差过大
FOR i:=1 TO g_setupJntNum BY 1 DO
	m_checkDelay[i_ArmId].T_armJntFollowErr[i](IN:= ABS(i_setupJointData.m_cmdJntPos[i_armId][i]- i_setupJointData.m_curJntPos[i_armId][i])>g_armMaxJntFollowErr[i]  AND m_checkPermit[i_ArmId].m_armJntFollowErr[i], PT:=m_checkDelayTime.Ti_armJntFollowErr , Q=> , ET=> );
	IF m_checkDelay[i_ArmId].T_armJntFollowErr[i].Q THEN
		errCodeAssign(i_ArmId, i_ArmId+3,  0, i, 16#2002, m_rcvLevel );
	END_IF
END_FOR


//关节速度监控
FOR i:=1 TO g_setupJntNum BY 1 DO
	m_checkDelay[i_ArmId].T_jntVelErr[i](IN:= ABS (i_setupJointData.m_curJntVel[i_armId][i])>g_safetyJntVel[i] AND m_checkPermit[i_ArmId].m_jntVelErr[i], PT:=m_checkDelayTime.Ti_jntVelErr , Q=> , ET=> );
	IF m_checkDelay[i_ArmId].T_jntVelErr[i].Q THEN
		errCodeAssign(i_ArmId, i_ArmId+3,  0, i, 16#2003, m_rcvLevel );
	END_IF
END_FOR



//电流超限监测
FOR i:=1 TO g_setupJntNum BY 1 DO
	m_checkDelay[i_ArmId].T_jntCurrentErr[i](IN:= ABS(i_setupJointData.m_rawJntCurrent[i_armId][i])>g_maxJntCurrent[i] AND m_checkPermit[i_ArmId].m_jntCurrentErr[i], PT:=m_checkDelayTime.Ti_jntCurrentErr , Q=> , ET=> );
	IF m_checkDelay[i_ArmId].T_jntCurrentErr[i].Q THEN
		errCodeAssign(i_ArmId, i_ArmId+3,  0, i, 16#2005, m_rcvLevel );
	END_IF
END_FOR


//Ethercat通讯检测
FOR i:=1 TO g_setupJntNum BY 1 DO
	IF NOT i_safetyCheckVar[i_ArmId].m_EtherCATState[i].EtherCATState THEN
		errCodeAssign(i_ArmId, i_ArmId+3, 0, i, 16#2006, m_rcvLevel );
	END_IF
END_FOR


//不动点发生变化监控
m_checkDelay[i_ArmId].T_FixedPointErr(IN:=  i_safetyCheckVar[i_ArmId].m_rcpCheck AND m_checkPermit[i_ArmId].m_fixedPointErr, PT:=m_checkDelayTime.Ti_FixedPointErr , Q=> , ET=> );
IF m_checkDelay[i_ArmId].T_FixedPointErr.Q THEN
	errCodeAssign(i_ArmId, i_ArmId+3,  0, 0, 16#2007, m_rcvLevel );
END_IF


//目标位置指令突变检测
FOR i:=1 TO g_setupJntNum BY 1 DO
	IF (i_setupJointData.m_cmdJntPos[i_armId][i]-m_cmdJntPosLast[i_ArmId][i])>g_maxJntCmdSalta[i] AND m_checkPermit[i_ArmId].m_cmdJntSaltation[i] THEN
		errCodeAssign(i_armId, i_ArmId+3, 0, i, 16#2008, m_rcvLevel );
	END_IF
	m_cmdJntPosLast[i_armId][i] := i_setupJointData.m_cmdJntPos[i_armId][i];
END_FOR


//Deviation between command current and feedback current
FOR i:=1 TO g_setupJntNum BY 1 DO
	IF ABS(i_safetyCheckVar[i_armId].m_slaveDriverOutput[i].m_cmdCurrent-i_safetyCheckVar[i_armId].m_slaveDriverInput[i].m_current)> g_jntCurrentCtrlLimit[i]  AND m_checkPermit[i_armId].m_jntCurrentCtrlErr[i] THEN
		//errCodeAssign(i_armId, i_armId+3, 0, i, 16#200B, m_rcvLevel );
	END_IF
END_FOR


//motor encoder mutation detection
FOR i:=1 TO g_setupJntNum BY 1 DO
	IF (i_safetyCheckVar[i_armId].m_motorEncoderSaltaValue[i])>g_maxJntCurSalta[i] THEN
		errCodeAssign(i_armId, i_ArmId+3, 0, i, 16#200C, m_rcvLevel );
	END_IF
END_FOR
END_METHOD

METHOD slaveSafetyCheck : BOOL
VAR_INPUT
	i_armId:UDINT;
	i_safetyCheckVar :ARRAY[1..g_maxNum] OF checkInputVariable;
	i_slaveJointData : ST_SlaveJointData;
END_VAR
//驱动器状态监测、驱动器未连接
FOR i:=1 TO g_sJntNum BY 1 DO
	m_checkDelay[i_ArmId].T_jntStatusErr[i+g_setupJntNum](IN:= (i_safetyCheckVar[i_ArmId].m_slaveDriverInput[i].m_statusWord=0 AND m_checkPermit[i_ArmId].m_jntStatusErr[i+g_setupJntNum]), PT:=m_checkDelayTime.Ti_jntStatusErr , Q=> , ET=> );
	IF m_checkDelay[i_ArmId].T_jntStatusErr[i+g_setupJntNum].Q  THEN
		errCodeAssign(i_ArmId, i_ArmId+3,  0, i+g_setupJntNum, 16#3002 ,m_unrcvLevel );
	END_IF
END_FOR



//关节编码器监测
FOR i:=1 TO g_sJntNum BY 1 DO
	m_checkDelay[i_ArmId].T_linkEncErr[i+g_setupJntNum](IN:= (i_safetyCheckVar[i_ArmId].m_slaveDriverInput[i].m_linkEncoder=g_maxLinkEnc[i] OR i_safetyCheckVar[i_ArmId].m_slaveDriverInput[i].m_linkEncoder=g_minLinkEnc[i]) AND m_checkPermit[i_ArmId].m_linkEncErr[i], PT:=m_checkDelayTime.Ti_linkEncErr , Q=> , ET=> );
	IF m_checkDelay[i_ArmId].T_linkEncErr[i+g_setupJntNum].Q THEN
		errCodeAssign(i_ArmId, i_ArmId+3,  0, i+g_setupJntNum,  16#3003 ,m_unrcvLevel );
	END_IF
END_FOR


//驱动器错误检测
FOR i:=1 TO g_sJntNum BY 1 DO
	m_checkDelay[i_ArmId].T_DriveErr[i+g_setupJntNum](IN:= (i_safetyCheckVar[i_ArmId].m_slaveDriverInput[i].m_driverError AND 16#20)=g_driveErrWord AND m_checkPermit[i_ArmId].m_driveErr[i] , PT:=m_checkDelayTime.Ti_driveErr , Q=> , ET=> );
	IF m_checkDelay[i_ArmId].T_DriveErr[i+g_setupJntNum].Q THEN
		errCodeAssign(i_ArmId, i_ArmId+3,  0, i+g_setupJntNum, 16#3004 ,m_unrcvLevel );
	END_IF
END_FOR


//双编码器偏差过大检测
FOR i:=1 TO g_sJntNum-5 BY 1 DO
	m_checkDelay[i_ArmId].T_armJntEncErr[i+g_setupJntNum](IN:= ABS(i_slaveJointData.m_curLinkPos[i_armId][i]-i_slaveJointData.m_curJntPos[i_armId][i])>=g_armMaxJntEncErr[i+g_setupJntNum] AND m_checkPermit[i_ArmId].m_armJntEncErr[i+g_setupJntNum], PT:=m_checkDelayTime.Ti_armJntEncErr , Q=> , ET=> );
	IF m_checkDelay[i_ArmId].T_armJntEncErr[i+g_setupJntNum].Q THEN
		errCodeAssign( i_ArmId, i_ArmId+3,  0, i+g_setupJntNum, 16#3005, m_unrcvLevel );
	END_IF
END_FOR


//关节运动超限位
FOR i:=1 TO g_sJntNum BY 1 DO
	m_checkDelay[i_ArmId].T_outOfLimit[i+g_setupJntNum](IN:= (i_slaveJointData.m_curJntPos[i_armId][i]>=(g_maxJntPos[i_armId,i+g_setupJntNum]+g_armJntPosLimitBuffer[i+g_setupJntNum]) OR i_slaveJointData.m_curJntPos[i_armId][i]<=(g_minJntPos[i_armId,i+g_setupJntNum]-g_armJntPosLimitBuffer[i+g_setupJntNum])) AND m_checkPermit[i_ArmId].m_outOfLimit[i+g_setupJntNum] , PT:=m_checkDelayTime.Ti_outofLimit , Q=> , ET=> );
	IF m_checkDelay[i_ArmId].T_outOfLimit[i+g_setupJntNum].Q THEN
		errCodeAssign(i_ArmId, i_ArmId+3,  0, i+g_setupJntNum, 16#3006, m_unrcvLevel );
	END_IF
END_FOR


//电机电角度偏差
FOR i:=1 TO g_sJntNum BY 1 DO
	IF ABS(electriAngleDev(i_safetyCheckVar[i_armId].m_slaveDriverInput[i].m_electriAngleDev))> g_motPhieErrLimit  AND m_checkPermit[i_ArmId].m_motPhieErr[i+g_setupJntNum] THEN
		errCodeAssign(i_ArmId, i_ArmId+3,  0, i+g_setupJntNum, 16#3008, m_unrcvLevel );
	END_IF
END_FOR


//驱动器内部通讯错误
FOR i:=1 TO g_sJntNum BY 1 DO
	m_checkDelay[i_ArmId].T_currentIsNotUpdate[i+g_setupJntNum](IN:= (i_safetyCheckVar[i_ArmId].m_slaveDriverInput[i].m_current=m_curJntTorqueIOlast[i_ArmId][i+g_setupJntNum] AND m_checkPermit[i_ArmId].m_currentIsNotUpdate[i+g_setupJntNum]), PT:=m_checkDelayTime.Ti_currentIsNotUpdate , Q=> , ET=> );
	IF  m_checkDelay[i_ArmId].T_currentIsNotUpdate[i+g_setupJntNum].Q THEN
		//errCodeAssign(i_ArmId, i_ArmId+3,  0, i+g_setupJntNum, 16#3009 ,m_unrcvLevel );
	END_IF
	m_curJntTorqueIOlast[i_ArmId][i+g_setupJntNum]:=i_safetyCheckVar[i_ArmId].m_slaveDriverInput[i].m_current;
END_FOR


//关节跟随误差过大
FOR i:=1 TO g_sJntNum BY 1 DO
	m_checkDelay[i_ArmId].T_armJntFollowErr[i+g_setupJntNum](IN:= ABS(i_slaveJointData.m_cmdJntPos[i_armId][i]- i_slaveJointData.m_curJntPos[i_armId][i])>g_armMaxJntFollowErr[i+g_setupJntNum]  AND m_checkPermit[i_ArmId].m_armJntFollowErr[i+g_setupJntNum], PT:=m_checkDelayTime.Ti_armJntFollowErr , Q=> , ET=> );
	IF m_checkDelay[i_ArmId].T_armJntFollowErr[i+g_setupJntNum].Q THEN
		errCodeAssign(i_ArmId, i_ArmId+3,  0, i+g_setupJntNum, 16#2002, m_rcvLevel );
	END_IF
END_FOR


//关节速度监控
FOR i:=1 TO g_sJntNum-5 BY 1 DO
	m_checkDelay[i_ArmId].T_jntVelErr[i+g_setupJntNum](IN:= ABS (i_slaveJointData.m_curJntVel[i_armId][i])>g_safetyJntVel[i+g_setupJntNum] AND m_checkPermit[i_ArmId].m_jntVelErr[i+g_setupJntNum], PT:=m_checkDelayTime.Ti_jntVelErr , Q=> , ET=> );
	IF m_checkDelay[i_ArmId].T_jntVelErr[i+g_setupJntNum].Q THEN
		errCodeAssign(i_ArmId, i_ArmId+3,  0, i+g_setupJntNum, 16#2003, m_rcvLevel );
	END_IF
END_FOR


// TODO: replaced with cartesin twist check
//笛卡尔空间指令与位置偏差检测
//FOR i:=1 TO 6 BY 1 DO
//	m_checkDelay[i_ArmId].T_spacePoseErr[i](IN:= i_safetyCheckVar[i_ArmId].m_spacePoseErr[i]> g_maxCartPoseErr[i] AND m_checkPermit[i_ArmId].m_spacePoseErr[i], PT:=m_checkDelayTime.Ti_spacePoseErr , Q=> , ET=> );
//	IF m_checkDelay[i_ArmId].T_spacePoseErr[i].Q THEN
//		errCodeAssign(i_ArmId, i_ArmId+3, 1, i, 16#2004, m_rcvLevel );
//	END_IF
//END_FOR


//电流超限监测
FOR i:=1 TO g_sJntNum BY 1 DO
	m_checkDelay[i_ArmId].T_jntCurrentErr[i+g_setupJntNum](IN:= ABS(i_slaveJointData.m_rawJntCurrent[i_armId][i])>g_maxJntCurrent[i+g_setupJntNum] AND m_checkPermit[i_ArmId].m_jntCurrentErr[i+g_setupJntNum], PT:=m_checkDelayTime.Ti_jntCurrentErr , Q=> , ET=> );
	IF m_checkDelay[i_ArmId].T_jntCurrentErr[i+g_setupJntNum].Q THEN
		errCodeAssign(i_ArmId, i_ArmId+3,  0, i+g_setupJntNum, 16#2005, m_rcvLevel );
	END_IF
END_FOR


//Ethercat通讯检测
FOR i:=1 TO g_sJntNum BY 1 DO
	IF NOT i_safetyCheckVar[i_ArmId].m_EtherCATState[i+g_setupJntNum].EtherCATState THEN
		errCodeAssign(i_ArmId, i_ArmId+3, 0, i+g_setupJntNum, 16#2006, m_rcvLevel );
	END_IF
END_FOR


//目标位置指令突变检测
FOR i:=1 TO g_sJntNum BY 1 DO
	m_checkDelay[i_ArmId].T_jntCmdSalta[i+g_setupJntNum](IN:= m_checkPermit[i_ArmId].m_cmdJntSaltation[i+g_setupJntNum], PT:=m_checkDelayTime.Ti_jntCmdSaltationErr , Q=> , ET=> );
	IF m_checkDelay[i_ArmId].T_jntCmdSalta[i+g_setupJntNum].Q THEN
		IF (i_slaveJointData.m_cmdJntPos[i_armId][i]-m_cmdJntPosLast[i_ArmId][i+g_setupJntNum])>g_maxJntCmdSalta[i+g_setupJntNum] THEN
			errCodeAssign(i_ArmId, i_ArmId+3, 0, i+g_setupJntNum, 16#2008, m_rcvLevel );
		END_IF
	END_IF
	m_cmdJntPosLast[i_ArmId][i+g_setupJntNum] := i_slaveJointData.m_cmdJntPos[i_armId][i];
END_FOR


//Deviation between command current and feedback current
//FOR i:=1 TO g_sJntNum BY 1 DO
//	IF ABS(i_safetyCheckVar[i_armId].m_slaveDriverOutput[i].m_cmdCurrent-i_safetyCheckVar[i_armId].m_slaveDriverInput[i].m_current)> g_jntCurrentCtrlLimit[i+g_setupJntNum]  AND m_checkPermit[i_armId].m_jntCurrentCtrlErr[i+g_setupJntNum] THEN
//		errCodeAssign(i_armId, i_armId+3, 0, i+g_setupJntNum, 16#200B, m_rcvLevel );
//	END_IF
//END_FOR


//motor encoder mutation detection
FOR i:=1 TO g_sJntNum BY 1 DO
	IF (i_safetyCheckVar[i_armId].m_motorEncoderSaltaValue[i+g_setupJntNum])>g_maxJntCurSalta[i+g_setupJntNum] THEN
		errCodeAssign(i_armId, i_ArmId+3, 0, i+g_setupJntNum, 16#200C, m_rcvLevel );
	END_IF
END_FOR


//器械张开角度过大或过小
IF (i_safetyCheckVar[i_ArmId].m_instruOpenAngle> g_maxInstruOpen OR i_safetyCheckVar[i_ArmId].m_instruOpenAngle< 0) AND m_checkPermit[i_ArmId].m_instruOpenAngle THEN
	errCodeAssign(i_ArmId, i_ArmId+3, 0, 0, 16#200D, m_rcvLevel );
END_IF
END_METHOD

METHOD systemSafetyCheck : BOOL
VAR_INPUT
	i_armId:UDINT;
	i_safetyCheckVar :ARRAY[1..g_maxNum] OF checkInputVariable;
	i_cartJointData : ST_CartJointData;
	i_setupJointData : ST_SetupJointData;
	i_slaveJointData : ST_SlaveJointData;
END_VAR

VAR
	k:INT;
END_VAR

IF i_armId =g_cartNum THEN 
	//cart safrty check
	cartSafetyCheck(i_armId,i_safetyCheckVar[i_armId],i_cartJointData);
ELSE
	//EmergencyStopButton
	IF NOT i_safetyCheckVar[i_ArmId].EmergencyStop OR m_jntErrFlag[i_armId,0,3] THEN
		errCodeAssign(i_ArmId, 16#0C, 0, 0, 16#3001, m_unrcvLevel);
		RETURN;
	END_IF
	//setup arms safety check
	setupSafetyCheck(i_armId,i_safetyCheckVar,i_setupJointData);
	//slave arms safety check
	slaveSafetyCheck(i_armId,i_safetyCheckVar,i_slaveJointData);
END_IF

//StopButton
IF NOT i_safetyCheckVar[i_ArmId].SlaveStopButton OR i_safetyCheckVar[i_ArmId].PCStopButton=0 OR i_safetyCheckVar[i_ArmId].MasterStopButton THEN
	errCodeAssign(i_ArmId, 16#0C, 0, 0, 16#2001, m_rcvLevel );
END_IF

//prompt message
FOR i:=1 TO 30 BY 1 DO
	PromptMassCode( i_safetyCheckVar[i_ArmId].m_promptStatus[i], i_ArmId,  i,  i_safetyCheckVar[i_ArmId].m_promptLocation[i]);
END_FOR
END_METHOD

METHOD vecDeleteInput : BOOL
VAR_IN_OUT CONSTANT
	vecA :ARRAY[*] OF UDINT;
END_VAR

VAR_INPUT
	i_deleteCode :UDINT;
END_VAR

VAR_IN_OUT
	vecB : ARRAY[*] OF UDINT;
END_VAR

VAR
	m :DINT;
	i :DINT;
	Falg:BOOL;
END_VAR
m:=UPPER_BOUND(vecA,1);

FOR i:=0 TO m BY 1 DO 
	IF vecA[i]=i_DeleteCode THEN
		Falg:=TRUE;
	END_IF
	
	IF Falg=TRUE THEN
		vecB[i]:=vecA[i+1];
	ELSE
		vecB[i]:=vecA[i];
	END_IF
END_FOR
vecB[m]:=0;
END_METHOD

METHOD vecFIFO : BOOL
VAR_IN_OUT CONSTANT
	vecA :ARRAY[*] OF UDINT;
END_VAR

VAR_INPUT
	i_newData :UDINT;
END_VAR

VAR_IN_OUT
	vecB : ARRAY[*] OF UDINT;
END_VAR

VAR
	m :DINT;
	i :DINT;
END_VAR
m:=UPPER_BOUND(vecA,1);

FOR i:=0 TO m DO
	vecB[i+1]:=vecA[i];
END_FOR

vecB[0]:=i_newData;
END_METHOD

END_FUNCTION_BLOCK

// ---- Mains/CartControl.TcPOU
PROGRAM CartControl
VAR
	// cart instance
	m_cartRobot :FB_CartRobot;
	
	// Output cart status
	m_cartStatus AT%Q* : ST_CartStatus;
	
	// cart joint data
	m_cartJointsData AT %Q* :ST_CartJointData;
	
	m_cartDataPool: ST_CartInputDataPool;
	
	// wait time before cart init for ethercat to be statble 
	m_cartInitWaitTime : LREAL:=0;
	
	// cart init flag
	m_cartInit :BOOL :=FALSE;
	
	m_workHeartTon0 : TON;
	m_workHeartTon1 : TON;
	m_dumpEnergy : UINT:=51;
	m_cartInSterileStateTon :Ton;
	m_cartInSterileState :BOOL;
	//Aseptic sleeve is installed flag
	m_asepticInstalledFlag : Vec4b;
	m_slaveArmDisableFlag : Vec4b;
END_VAR

// wait communication to be stable
IF(m_cartInitWaitTime<g_robotInitWaitTime) THEN
	m_cartInitWaitTime := m_cartInitWaitTime+g_cartCtrlCycleTime;
	RETURN;
END_IF

// cart init
IF m_cartInit =FALSE THEN
	m_cartRobot.Init();
	m_cartInit:=TRUE;
END_IF

// input from UI
UIInputProcess();

// cart run
m_cartRobot.run(m_cartDataPool);

m_cartRobot.getStatus(m_cartStatus,m_cartJointsData);


UIOutputProcess();

// tranform data from UI(global variable write by ADS) to ST_UIData
METHOD UIInputProcess : BOOL
VAR_INPUT
END_VAR
VAR
	i:int;
END_VAR
// cart Joystick data
m_cartDataPool.m_UIData.m_joystickDataFromUI := GVL_interactUI.g_joystickSignalArray;

m_cartDataPool.m_UIData.m_ctrlEnableFromUI := GVL_interactUI.g_uiCtrl;

//limit_height:UINT;  上位机的高度值单位是mm，系统的高度值单位是m，底座高度是1805mm
//打开ui_control.limit_height_adjusting后可以调整立柱，并实时将立柱当前高度上传
IF (GVL_interactUI.g_uiCtrl.m_heightLimitAdjustEnable=TRUE) THEN
	m_cartDataPool.m_UIData.m_standColumnHightLimit := GVL_CartMotorParameters.g_maxJntPos[5];
ELSIF  (GVL_interactUI.g_uiCtrl.m_heightLimitAdjustEnable=FALSE) AND GVL_interactUI.g_heightLimitEnbale AND ABS((m_cartDataPool.m_UIData.m_standColumnHightLimit *1000+1850)-GVL_interactUI.g_heightLimitFromUI)>5 THEN
	m_cartDataPool.m_UIData.m_standColumnHightLimit := UINT_TO_LREAL(GVL_interactUI.g_heightLimitFromUI-GVL_CartControlParameters.g_cartInitialHeight)/1000;
ELSIF GVL_interactUI.g_heightLimitEnbale=FALSE THEN
	m_cartDataPool.m_UIData.m_standColumnHightLimit := GVL_CartMotorParameters.g_maxJntPos[5];
END_IF
GVL_interactUI.g_heightLimit :=LREAL_TO_UINT (m_cartRobot.m_slaveCart.curJntPos[5] * 1000 + GVL_CartControlParameters.g_cartInitialHeight);

//Surgical orientation selection
m_cartDataPool.m_UIData.m_surgicalSite := GVL_interactUI.g_surgicalSite;
m_cartDataPool.m_UIData.m_surgicalLocation := GVL_interactUI.g_surgicalLocation;

m_dumpEnergy := GVL_interactUI.g_dumpEnergyUPS;
END_METHOD

METHOD UIOutputProcess : BOOL
VAR_INPUT
END_VAR
VAR 
	i : INT;
END_VAR
//TODO
//work heart
m_workHeartTon0(IN:= GVL_interactUI.g_heartBeat = 1, PT:= T#1S, Q=> , ET=> );
m_workHeartTon1(IN:= GVL_interactUI.g_heartBeat = 0, PT:= T#1S, Q=> , ET=> );
IF m_workHeartTon0.Q THEN
	GVL_interactUI.g_heartBeat :=0 ;
ELSIF m_workHeartTon1.Q THEN
	GVL_interactUI.g_heartBeat  :=1 ;
END_IF

GVL_interactUI.g_cartOperation.m_drapingAdjustState := m_cartRobot.m_slaveCart.m_cartDataFromUI.m_cartDrapingState;
GVL_interactUI.g_cartOperation.m_dockingAdjustState := m_cartRobot.m_slaveCart.m_cartDataFromUI.m_cartDockingState;

GVL_interactUI.g_trocarStatus := INT_TO_BOOL(m_cartRobot.m_slaveCart.m_trocarOnFlag);

GVL_interactUI.g_slaveRunAlone := NOT SlaveArmControl.m_slaveRobot.m_masterOnLine;
GVL_interactUI.g_joysticksTrigger := SafetyCheck.m_joysticksTrigger;

IF GVL_interactUI.g_surgicalStatus = 1 THEN
	IF NOT SlaveArmControl.m_slaveRobotData.m_asepticDeployCompletedFlag THEN
		m_slaveArmDisableFlag := g_zeroVec4b;
	END_IF
	GVL_interactUI.g_cartOperation.m_setupSterileState := BOOL_TO_UINT(m_asepticInstalledFlag[1]) OR BOOL_TO_UINT(m_asepticInstalledFlag[2]) OR BOOL_TO_UINT(m_asepticInstalledFlag[3]) OR BOOL_TO_UINT(m_asepticInstalledFlag[4]) ;
ELSE
	GVL_interactUI.g_cartOperation.m_setupSterileState := BOOL_TO_UINT(m_asepticInstalledFlag[1]) AND BOOL_TO_UINT(m_asepticInstalledFlag[2]) AND BOOL_TO_UINT(m_asepticInstalledFlag[3]) AND BOOL_TO_UINT(m_asepticInstalledFlag[4]) ;
	m_slaveArmDisableFlag := SlaveArmControl.m_slaveInputDataPool.m_UIData.m_slaveArmDisableFlag;	
END_IF

FOR i := 1 TO 4 BY 1 DO
	m_asepticInstalledFlag[i] := m_slaveArmDisableFlag[i] OR SlaveArmControl.m_slaveRobot.m_panelMountedFlag[i];
END_FOR

GVL_interactUI.g_cartOperation.m_setupSterileStateArm1 := BOOL_TO_UINT(m_asepticInstalledFlag[1]); 
GVL_interactUI.g_cartOperation.m_setupSterileStateArm2 := BOOL_TO_UINT(m_asepticInstalledFlag[2]); 
GVL_interactUI.g_cartOperation.m_setupSterileStateArm3 := BOOL_TO_UINT(m_asepticInstalledFlag[3]); 
GVL_interactUI.g_cartOperation.m_setupSterileStateArm4 := BOOL_TO_UINT(m_asepticInstalledFlag[4]); 

GVL_interactUI.g_cartOperation.m_scopeInstalled := BOOL_TO_UINT(m_cartDataPool.m_slaveStatus.m_endoscopeMounted);

FOR i := 1 TO 4 BY 1 DO
	IF SlaveArmControl.m_slaveRobot.m_slaveArms[i].instrument.Instrutype<>InstruType_endoscope THEN
		IF SlaveArmControl.m_slaveRobot.m_instrumentMountedFlag[i] AND SlaveArmControl.m_slaveRobot.m_endoscopeMounted THEN
			GVL_interactUI.g_cartOperation.m_inSurgicalAllowed := 1;
			EXIT;
		ELSE
			GVL_interactUI.g_cartOperation.m_inSurgicalAllowed := 0;
		END_IF	
	END_IF	
END_FOR


//Cart_static_in_sterile_state:UINT; //台车进入无菌区，并且台车停止运动(连续10s没有运动)，0：没有完成，1：完成
IF m_cartRobot.m_slaveCart.m_cartDataFromUI.m_cartDockingState = 1 THEN
	IF m_cartRobot.m_CartState = CartJointState_Movement THEN
		m_cartInSterileState := FALSE;
	ELSIF m_cartRobot.m_lastCartState = CartJointState_Movement THEN
		m_cartInSterileState := TRUE;
	END_IF
ELSE
	m_cartInSterileState := FALSE;
	GVL_interactUI.g_cartOperation.m_cartInSterileState:=0;
END_IF
m_cartInSterileStateTon(IN:= m_cartInSterileState, PT:= T#10S, Q=> , ET=> );
IF m_cartInSterileStateTon.Q THEN
	GVL_interactUI.g_cartOperation.m_cartInSterileState:=1;
END_IF
END_METHOD

END_PROGRAM

// ---- FBs_Robots/FB_CartRobot.TcPOU
FUNCTION_BLOCK FB_CartRobot
VAR_INPUT
END_VAR
VAR_OUTPUT
END_VAR
VAR

	m_slaveCart: FB_SlaveCart;		
	
	// input arm button 
	m_carHandChassisDriveUnlock AT%I* :ARRAY [1..2] OF BOOL;
	
	//open laser io
	m_openHorizonLaser AT  %Q* :DINT;
	m_openCrossLaser AT  %Q* :DINT;

	m_joystickData:Vec8d;

	// all cart controller instance 
	m_cartCtrlFactory :ARRAY[1..CartJointState_totalNum] OF I_CartJointCtrl;
	
	m_cartState:E_CartJointState:=CartJointState_Init;
	m_lastCartState:E_CartJointState:=CartJointState_Init;
	m_nextCartState:E_CartJointState:=CartJointState_Init;
	
	// flag if cart joint self-check passed
	m_selfCheckPass:  BOOL :=FALSE;
	
	// all cart controller instance 
	m_cartError :FB_CartCtrlError;
	m_cartInit :FB_CartCtrlInit;
	m_cartReady :FB_CartCtrlReady;
	m_cartInSurgery :FB_CartCtrlInSurgery;
	m_cartMotionCar :FB_CartCtrlMotionCar;
	m_cartAsepticDeploy :FB_CartCtrlAsepticDeploy;
	m_cartAdjust :FB_CartCtrlAdjust;
	m_cartRotaOverhang :FB_CartCtrlRotaOverhang;
	m_cartSlowStop : FB_CartCtrlSlowDown;
	m_cartStandColuAdjust : FB_CartCtrlStandColuAdjust;
	m_cartSupporLeg : FB_CartSupporLeg;
	
	// cart controller interface
	m_cartCtrl : I_CartJointCtrl;
	m_cartCtrlCmds : ST_SlaveArmCtrlCmds;
	
	//state machine flow jump condition allowed
	m_hangAdjustAllowed : BOOL;
	m_asepticDeploymentAllowed :BOOL;
	m_cartMoveAllowed :BOOL;
	m_rotaOverhangAllowed :BOOL;
END_VAR

METHOD getStatus : BOOL
VAR_IN_OUT
	
	r_cartStatus :ST_CartStatus;	

	// cart joint data
	r_cartJointsData :ST_CartJointData;
END_VAR

VAR 
	i : INT;
END_VAR
r_cartStatus.m_CartState :=m_cartState;

r_cartStatus.m_uiControl := GVL_interactUI.g_uiCtrl;
r_cartStatus.m_cartDumpEnergy := GVL_interactUI.g_dumpEnergyUPS;
r_cartStatus.m_sdrivingLeverSensorManualFlag :=NOT m_slaveCart.m_drivingLeverSensorManual;
//r_cartStatus.m_stabilizerDeployedFlag
r_cartStatus.m_trocarOnFlag := m_slaveCart.m_trocarOnFlag;
r_cartStatus.m_joystickValue := m_slaveCart.m_joystickSignal;
r_cartStatus.m_jntPosReachLimit := m_cartAdjust.jntPosReachLimit;

r_cartJointsData.m_cmdJntPos := m_slaveCart.cmdJntPos;
r_cartJointsData.m_cmdJntVel := m_slaveCart.cmdJntVel;
r_cartJointsData.m_curJntPos := m_slaveCart.curJntPos;
r_cartJointsData.m_curJntTrq := m_slaveCart.curJntCurrent;
r_cartJointsData.m_curJntVel := m_slaveCart.curJntVel;
r_cartJointsData.m_curLinkPos := m_slaveCart.curLinkPos;
r_cartJointsData.m_curMotorPos := m_slaveCart.curMotorPos;
END_METHOD

METHOD init : BOOL
VAR_INPUT
END_VAR
VAR
	i:INT;
END_VAR

m_slaveCart.init();
m_cartState := CartJointState_Init;
m_lastCartState := CartJointState_Init;
m_nextCartState := CartJointState_Init;
m_selfCheckPass := FALSE;

//command init
m_cartCtrlCmds.m_jntEnableFlag := g_zeroVec8i;
m_cartCtrlCmds.m_jntOPMode := g_slaveAllPosMode;
m_cartCtrlCmds.m_cmdJntPos := m_slaveCart.m_curJntPos;
m_cartCtrlCmds.m_cmdJntVel := g_zeroVec8d;
m_cartCtrlCmds.m_cmdJntAcc := g_zeroVec8d;
m_cartCtrlCmds.m_cmdJntTrq := g_zeroVec8d;


// generate controller factory
//m_cartCtrlFactory[CartJointState_Error] := m_cartError;
m_cartCtrlFactory[CartJointState_Init] := m_cartInit;
m_cartCtrlFactory[CartJointState_Ready] := m_cartReady;
m_cartCtrlFactory[CartJointState_InSurgery] := m_cartInSurgery;
m_cartCtrlFactory[CartJointState_Movement] := m_cartMotionCar;
m_cartCtrlFactory[CartJointState_HangAdjust] := m_cartAdjust;
m_cartCtrlFactory[CartJointState_AsepticDeployment] := m_cartAsepticDeploy;
m_cartCtrlFactory[CartJointState_RotaOverhang] := m_cartRotaOverhang;
m_cartCtrlFactory[CartJointState_SlowStop] := m_cartSlowStop;
m_cartCtrlFactory[CartJointState_StandColuAdjust] := m_cartStandColuAdjust;
m_cartCtrlFactory[CartJointState_SupporLeg] := m_cartSupporLeg;

// assign controller
m_cartCtrl:=m_cartCtrlFactory[m_cartState];
m_cartCtrl.Init(m_slaveCart,m_cartCtrlCmds);
END_METHOD

METHOD laserIO : BOOL
VAR_INPUT
END_VAR

//cross laser IO output , when slave self check succeed , and trocar  install at least one
IF GVL_interactUI.g_slaveSelfCheckStatus = 2 AND m_slaveCart.m_trocarOnFlag = 0 THEN
	m_openCrossLaser := 1;
ELSE
	m_openCrossLaser := 0;
END_IF

//Horizontal laser IO output ,when adjusting the trolley or moving the trolley
IF (m_slaveCart.curJntPos[5] * 1000 + GVL_CartControlParameters.g_cartInitialHeight) > GVL_CartControlParameters.g_cartOpenHorizonLaserHeight AND  (m_cartState = CartJointState_Movement OR m_cartState = CartJointState_HangAdjust) THEN
	m_openHorizonLaser :=  1;
ELSE
	m_openHorizonLaser :=  0;
END_IF
END_METHOD

METHOD PUBLIC run : BOOL
VAR_IN_OUT CONSTANT
	i_cartDataPool: ST_CartInputDataPool;
END_VAR
VAR
	i:INT;
END_VAR
// state machine transition
stateMachine(i_cartDataPool);	

//update ui data
m_slaveCart.ProcessingUIData(i_cartDataPool.m_UIData);

//update cart joint status
m_slaveCart.updateStatus();

laserIO();

// null ptr check
IF 0 = m_cartCtrl THEN
	RETURN;
END_IF

// run controller
m_cartCtrl.run(m_slaveCart,m_cartCtrlCmds);


m_slaveCart.updateCmds(m_cartCtrlCmds);
END_METHOD

METHOD PROTECTED stateMachine : BOOL
VAR_IN_OUT CONSTANT
	i_cartDataPool: ST_CartInputDataPool;
END_VAR
VAR
	i,j:INT;
END_VAR
m_hangAdjustAllowed := m_slaveCart.m_trocarOnFlag=0 AND ( i_cartDataPool.m_UIData.m_ctrlEnableFromUI.m_joystickEnable OR i_cartDataPool.m_UIData.m_ctrlEnableFromUI.m_cameraJoystickEnable);
m_asepticDeploymentAllowed := m_slaveCart.m_trocarOnFlag=0 AND ((i_cartDataPool.m_UIData.m_ctrlEnableFromUI.m_dockingEnable AND m_slaveCart.cartDockingState=0) 
												OR (i_cartDataPool.m_UIData.m_ctrlEnableFromUI.m_drapingEnable AND m_slaveCart.cartDrapingState=0)) AND NOT ( i_cartDataPool.m_safetyData.m_cartAdjustErr OR i_cartDataPool.m_safetyData.m_cartStandColumnErr) ;
m_cartMoveAllowed := m_slaveCart.m_trocarOnFlag=0 AND  (m_carHandChassisDriveUnlock[1] OR m_carHandChassisDriveUnlock[2]) AND NOT i_cartDataPool.m_safetyData.m_cartWheelErr;
m_rotaOverhangAllowed := m_slaveCart.m_trocarOnFlag=0 AND m_slaveCart.m_rotaOverhangOnFlag > 1 AND NOT i_cartDataPool.m_safetyData.m_cartOverhangErr;

// state machine transit
CASE m_cartState OF
	//cart joint error
	CartJointState_Error:
		//IF FALSE = i_cartDataPool.m_safetyData.m_slaveErrFlag THEN
		//	// to standby
		//	IF m_selfCheckPass THEN
		//		m_nextCartState :=CartJointState_Standby;
		//	ELSE
		//		m_nextCartState :=CartJointState_Init;
		//	END_IF
		//END_IF

	CartJointState_Init:
		IF m_cartCtrl.isFinished THEN
			m_nextCartState :=CartJointState_Ready;
		END_IF
		
		
	CartJointState_Ready:
		IF m_cartCtrl.isFinished  THEN
			m_nextCartState := CartJointState_InSurgery;
			
		ELSIF m_hangAdjustAllowed THEN
			m_nextCartState := CartJointState_HangAdjust;
			
		ELSIF m_asepticDeploymentAllowed THEN
			m_nextCartState := CartJointState_AsepticDeployment;
			
		ELSIF m_cartMoveAllowed THEN
			m_nextCartState := CartJointState_Movement;
			
		ELSIF m_rotaOverhangAllowed THEN
			m_nextCartState := CartJointState_RotaOverhang;
			
		ELSIF m_slaveCart.m_trocarOnFlag=0 AND  m_slaveCart.m_columnAdjustEnable  THEN
			m_nextCartState := CartJointState_StandColuAdjust;
		END_IF
		
	
	CartJointState_InSurgery:
		IF m_cartCtrl.isFinished  THEN
			m_nextCartState :=CartJointState_Ready;
		END_IF
		
		
	CartJointState_Movement:
		IF m_slaveCart.m_trocarOnFlag<>0 OR (NOT m_carHandChassisDriveUnlock[1] AND NOT m_carHandChassisDriveUnlock[2])  THEN
			m_nextCartState :=CartJointState_SlowStop;
		ELSIF i_cartDataPool.m_safetyData.m_cartWheelErr THEN
			m_nextCartState :=CartJointState_Ready;
		END_IF
		
		
	CartJointState_HangAdjust:
		IF  m_slaveCart.m_trocarOnFlag<>0 OR (NOT i_cartDataPool.m_UIData.m_ctrlEnableFromUI.m_joystickEnable AND NOT i_cartDataPool.m_UIData.m_ctrlEnableFromUI.m_cameraJoystickEnable ) THEN
			m_nextCartState :=CartJointState_SlowStop;
		END_IF
		
		
	CartJointState_AsepticDeployment:
		IF m_cartCtrl.isFinished  THEN
			IF i_cartDataPool.m_UIData.m_ctrlEnableFromUI.m_dockingEnable THEN
				m_slaveCart.cartDockingState := 1;
			ELSIF i_cartDataPool.m_UIData.m_ctrlEnableFromUI.m_drapingEnable THEN
				m_slaveCart.cartDrapingState := 1;
			END_IF
			m_nextCartState :=CartJointState_SlowStop;
		ELSIF i_cartDataPool.m_safetyData.m_cartAdjustErr OR i_cartDataPool.m_safetyData.m_cartStandColumnErr THEN
			m_nextCartState :=CartJointState_Ready;
		ELSIF m_slaveCart.m_trocarOnFlag<>0 OR (NOT i_cartDataPool.m_UIData.m_ctrlEnableFromUI.m_dockingEnable AND NOT i_cartDataPool.m_UIData.m_ctrlEnableFromUI.m_drapingEnable) THEN
			m_nextCartState :=CartJointState_SlowStop;
		END_IF
		
		
	CartJointState_RotaOverhang:
		IF m_slaveCart.m_rotaOverhangOnFlag <= 1 OR  m_slaveCart.m_trocarOnFlag<>0  THEN
			m_nextCartState :=CartJointState_SlowStop;
		ELSIF i_cartDataPool.m_safetyData.m_cartOverhangErr THEN
			m_nextCartState :=CartJointState_Ready;
		END_IF
		
	CartJointState_StandColuAdjust:
		IF (m_slaveCart.m_trocarOnFlag<>0 OR i_cartDataPool.m_safetyData.m_cartStandColumnErr) OR  NOT m_slaveCart.m_columnAdjustEnable  THEN
			m_nextCartState :=CartJointState_SlowStop;
		END_IF	
	
	CartJointState_SlowStop:
		IF m_cartCtrl.isFinished  THEN
			m_nextCartState :=CartJointState_Ready;
		END_IF
		
	CartJointState_SupporLeg:
		IF m_cartCtrl.isFinished  THEN
			m_nextCartState :=CartJointState_Ready;
		END_IF
END_CASE

// Controller transit
IF m_nextCartState<> m_cartState THEN
	//reset current controller
	m_cartCtrl.reset();
	
	// transit to new controller
	m_lastCartState:=m_cartState;
	m_cartState:=m_nextCartState;
	m_cartCtrl:=m_cartCtrlFactory[m_cartState];
	
	//init next controller
	m_cartCtrl.Init(m_slaveCart, m_cartCtrlCmds);
	m_slaveCart.updateCmds(m_cartCtrlCmds);
END_IF
END_METHOD

END_FUNCTION_BLOCK

// ---- FBs_Robots/FB_SlaveCart.TcPOU
FUNCTION_BLOCK FB_SlaveCart
VAR
	
	//Driving force of the car io
	m_driveForce AT %I* :ARRAY [1..6] OF DINT;
	
	//stabilizing foot sensor  (normally-closed contact)
	m_stabilizFootSensorLeft AT%I* :BOOL;
	m_stabilizFootSensorRight AT%I* :BOOL;
	m_drivingLeverSensorAuto AT%I* :BOOL;
	m_drivingLeverSensorManual AT%I* :BOOL;
	
	//Trocar IO check
	m_trocarIO AT %I* : ARRAY [1..4] OF UDINT;
	m_trocarCheck : ARRAY [1..4] OF FB_trocarDetect;
	m_trocarFlag : ARRAY [1..4] OF BOOL;
	m_trocarOnFlag : INT:=0;
	
	//output screw break IO 
	m_screwBreak AT %Q* : BOOL;
	m_screwBreakSR : SR;
	
	//car overhang rotation signal is in the arm
	m_carRotaOverhangIO AT%I* : ARRAY [1..4] OF UDINT;
	m_rotaButtonDetect : ARRAY [1..4] OF FB_rotaButtonDetect;
	m_rotaOverhangOnFlag : UDINT :=0;
	
	//cart joint
	m_cartJoints: ARRAY [1..g_cartJntNum] OF FB_CartJoint;
	
	// cart status
	m_cartStatus  : ST_CartStatus;
	
	//cart joint 5 enable detect
	m_standColumnEnableDetect : FB_cartJntEnableDetect;
	m_standColumnDisenableDetect : FB_cartJntDisenableDetect;

		// arm joint data
	m_curMotorPos :Vec8d;
	m_curLinkPos :Vec8d;
	m_curLinkSingle :Vec8d;
	m_curJntPos :Vec8d;
	m_curDHJntPos :Vec6d;
	m_curGripAngle :LREAL;
	m_curJntVel :Vec8d;
	m_curDHJntVel :Vec6d;
	m_curJntTrq :Vec8d;
	m_rawJntCurrent :Vec8d;
	m_filtJntCurrent :Vec8d;
	m_cmdJntTrq :Vec8d;
	m_cmdJntCurrent : Vec8d;
	m_cmdJntPos :Vec8d;
	m_cmdJntVel :Vec8d;

	//SDO Writer
	m_CommunicationCycleInitMZSub1:ARRAY [1..3] OF FB_EcCoESdoWrite;
	m_CommunicationCycleInitMZSub2:ARRAY [1..3] OF FB_EcCoESdoWrite;
	m_CommunicationCycleSub1:INT:=1;
	m_CommunicationCycleSub2:INT:=-3;
	
	//update ui information
	m_joystickSignalIO AT %I* : ARRAY [1..8] OF UDINT;
	m_joystickSignal : Vec8d;
	m_cartDataFromUI : ST_CartUIData;
	m_ctrlEnable : ST_uiControl;
	m_surgicalStatusF : F_TRIG;
	
	//stand column adjust of setup joint 3
	m_columnJntVel : LREAL;
	m_columnAdjustEnable : BOOL;
	m_limitBufferForCtrl : LREAL := 0.01;
	m_midJntPos : LREAL := 0.1;
	enableTon : ARRAY [1..4] OF FB_TON;
END_VAR

PROPERTY cartDockingState : UINT
GET
END_GET
SET
m_cartDataFromUI.m_cartDockingState := cartDockingState;
END_SET
END_PROPERTY

PROPERTY cartDrapingState : UINT
GET
END_GET
SET
m_cartDataFromUI.m_cartDrapingState := cartDrapingState;
END_SET
END_PROPERTY

METHOD checkIO : BOOL
VAR_INPUT
END_VAR
VAR
	i:INT;
END_VAR
//check overhang rotation button
m_rotaOverhangOnFlag := MAX( m_rotaButtonDetect[1].run(m_carRotaOverhangIO[1]), m_rotaButtonDetect[2].run(m_carRotaOverhangIO[2]),m_rotaButtonDetect[3].run(m_carRotaOverhangIO[3]),m_rotaButtonDetect[4].run(m_carRotaOverhangIO[4]));

FOR i := 1 TO g_sArmNum BY 1 DO
	//trocar in place monitor
	m_trocarFlag[i] := m_trocarCheck[i].run(m_trocarIO[i] );
END_FOR

m_trocarOnFlag := BOOL_TO_INT(m_trocarFlag[1]) + BOOL_TO_INT(m_trocarFlag[2]) + BOOL_TO_INT(m_trocarFlag[3]) + BOOL_TO_INT(m_trocarFlag[4]);

//setup robot joint 3 adjust and drive column movement
m_columnAdjustEnable :=columnAdjustEnable(o_columnJntVel => m_columnJntVel  );
END_METHOD

PROPERTY cmdJntPos : REFERENCE TO Vec8d
GET
cmdJntPos REF= m_cmdJntPos;
END_GET
END_PROPERTY

PROPERTY cmdJntVel : REFERENCE TO Vec8d
GET
cmdJntVel REF= m_cmdJntVel;
END_GET
END_PROPERTY

METHOD columnAdjustEnable : BOOL
VAR_INPUT
END_VAR

VAR_OUTPUT
	o_columnJntVel : LREAL;
END_VAR

VAR_STAT
	curJntPos : vec4d;
	curJntVel : vec4d;
	columnJntVel : vec4d;
	adjustStartFlag : vec4b;
	m_columnAdjustEnable : vec4b;
END_VAR
VAR
	i : INT;
	armId : INT;
	limitDis : vec4d;
	m_adjustFlag : vec4b;
END_VAR

FOR i := 1 TO g_sArmNum DO
	curJntPos[i] := SetupArmControl.m_setupRobot.m_setupArms[i].m_curJntPos[3];
	curJntVel[i] := SetupArmControl.m_setupRobot.m_setupArms[i].m_curJntVel[3];
	m_adjustFlag[i] := SetupArmControl.m_setupRobot.m_setupArms[i].m_manualAdjustOnFlag AND m_trocarOnFlag=0 AND SetupArmControl.m_setupRobot.m_setupArmState[i] = SetupArmState_ManualAdjust 
									AND NOT SafetyCheck.m_SafetyCheck.m_jntErrFlag[i,0,2] AND NOT SafetyCheck.m_SafetyCheck.m_jntErrFlag[i,0,3] AND NOT SafetyCheck.m_SafetyCheck.m_jntErrFlag[i,3,3] AND NOT SafetyCheck.m_SafetyCheck.m_jntErrFlag[i,2,3] ;
	
	IF m_adjustFlag[i] THEN
		limitDis[i] := MIN(GVL_SetupMotorParameters.g_maxJntPos[i,3] - curJntPos[i], curJntPos[i]-GVL_SetupMotorParameters.g_minJntPos[i,3]);
		IF limitDis[i] < m_limitBufferForCtrl THEN
			adjustStartFlag[i] := TRUE; 
			columnJntVel[i] := sign(m_midJntPos - curJntPos[i]) * GVL_CartControlParameters.g_maxJntVel[5];
		
		ELSIF limitDis[i] >= m_limitBufferForCtrl AND NOT m_columnAdjustEnable[i] THEN
			columnJntVel[i] := 0;
			adjustStartFlag[i] := FALSE;
			
		ELSE
			IF curJntVel[i] <> 0 AND adjustStartFlag[i] THEN
				columnJntVel[i] := -LIMIT(-GVL_CartControlParameters.g_maxJntVel[5], curJntVel[i], GVL_CartControlParameters.g_maxJntVel[5]);
			END_IF
		END_IF
		
		armId := i;
		enableTon[i](IN:= adjustStartFlag[i], PT:= T#3S, Q=> m_columnAdjustEnable[i], ET=> );
		EXIT;
	ELSE
		adjustStartFlag[i] := FALSE;
		columnJntVel[i] := 0;
	END_IF
	enableTon[i](IN:= adjustStartFlag[i], PT:= T#3S, Q=> m_columnAdjustEnable[i], ET=> );
END_FOR

//output stand column joint velocity and start adjust single
IF armId > 0 THEN
	o_columnJntVel := columnJntVel[armId];
END_IF
columnAdjustEnable := m_columnAdjustEnable[1] OR m_columnAdjustEnable[2] OR m_columnAdjustEnable[3] OR m_columnAdjustEnable[4];
END_METHOD

PROPERTY ctrlEnable : REFERENCE TO ST_uiControl
GET
ctrlEnable REF= m_ctrlEnable;
END_GET
SET
END_SET
END_PROPERTY

PROPERTY curDHJntPos :REFERENCE TO Vec6d
GET
curDHJntPos ref= m_curDHJntPos;
END_GET
END_PROPERTY

PROPERTY curDHJntVel :REFERENCE TO Vec6d
GET
curDHJntVel REF= m_curDHJntVel;
END_GET
END_PROPERTY

PROPERTY curJntCurrent :REFERENCE TO Vec8d
GET
curJntCurrent ref=m_filtJntCurrent;
END_GET
END_PROPERTY

PROPERTY curJntPos : REFERENCE TO Vec8d
GET
curJntPos ref=m_curJntPos;
END_GET
END_PROPERTY

PROPERTY curJntVel :REFERENCE TO Vec8d
GET
curJntVel ref=m_curJntVel;
END_GET
END_PROPERTY

PROPERTY curLinkPos :REFERENCE TO Vec8d
GET
curLinkPos ref=m_curLinkPos;
END_GET
END_PROPERTY

PROPERTY curMotorPos : REFERENCE TO  Vec8d
GET
curMotorPos ref=m_curMotorPos;
END_GET
END_PROPERTY

METHOD PUBLIC enable : BOOL
VAR_IN_OUT CONSTANT
	i_jntIdx :Vec8i;
END_VAR
VAR
	i :INT ;
END_VAR
FOR i:=1 TO g_cartJntNum DO
	IF 3<=i AND i<5 THEN
		IF 1= i_jntIdx[i] THEN
			m_cartJoints[i].enableMZ();
		ELSE
			m_cartJoints[i].disable();
		END_IF
	ELSIF i = 5 THEN
		IF 1= i_jntIdx[i] THEN
			m_screwBreak := m_standColumnEnableDetect.run(IOValue:= m_cartJoints[i].enableMZ());
			m_standColumnDisenableDetect.run(IOValue:=FALSE );
		ELSE
			m_standColumnEnableDetect.run(IOValue:= FALSE);
			m_screwBreak :=  NOT m_standColumnDisenableDetect.run(IOValue:=m_cartJoints[i].disable());
		END_IF
	ELSE
		IF 1= i_jntIdx[i] THEN
			m_cartJoints[i].enable();
		ELSE
			m_cartJoints[i].disable();
		END_IF
	END_IF
END_FOR
END_METHOD

METHOD init : BOOL
VAR_INPUT
END_VAR
VAR
	i:INT;
END_VAR


// cart joint init
FOR i:= 1 TO g_cartJntNum BY 1 DO
	m_cartJoints[i].init(i, g_cartCtrlCycleTime);
END_FOR


// joint init
FOR i:=1 TO g_cartJntNum DO
	m_cartJoints[i].initJntPos();
END_FOR


// update cart status if joint position is re-init
updateStatus();



//MingZhi drive example Initialize the communication period
FOR i := 1 TO 3 BY 1 DO
	m_CommunicationCycleInitMZSub1[i](sNetID:= GVL_CartJointEncoderCaliData.g_slaveCartNetID,
				nSlaveAddr := GVL_CartJointEncoderCaliData.g_slaveCartJointNetPort[i+2],
				nSubIndex:=1,nIndex:=16#60C2,pSrcBuf:=ADR(m_CommunicationCycleSub1),cbBufLen:=SIZEOF(m_CommunicationCycleSub1),bExecute:=TRUE);
	
	IF NOT m_CommunicationCycleInitMZSub1[i].bBusy THEN
		m_CommunicationCycleInitMZSub1[i](bExecute:=FALSE);
	END_IF
					
	m_CommunicationCycleInitMZSub2[i](sNetID:= GVL_CartJointEncoderCaliData.g_slaveCartNetID,
					nSlaveAddr := GVL_CartJointEncoderCaliData.g_slaveCartJointNetPort[i+2],
					nSubIndex:=2,nIndex:=16#60C2,pSrcBuf:=ADR(m_CommunicationCycleSub2),cbBufLen:=SIZEOF(m_CommunicationCycleSub2),bExecute:=TRUE);
	
	IF NOT m_CommunicationCycleInitMZSub2[i].bBusy THEN
		m_CommunicationCycleInitMZSub2[i](bExecute:=FALSE);
	END_IF
END_FOR
END_METHOD

METHOD  joystickSignalAnalysis : Vec8d 
VAR_INPUT
	//i_joystickDataFromUI:ARRAY [0..21] OF USINT;
	i_joystickDataFromUI:ARRAY [1..8] OF UDINT;
END_VAR

VAR_STAT
	i:INT;
	m_handData:ARRAY [1..8] OF UDINT;
	m_outHandData : Vec8d;
END_VAR

//IF i_joystickDataFromUI[0] = 16#FF THEN
//	m_handData := i_joystickDataFromUI;
//	m_outHandData[1] :=m_handData[7]*256 + m_handData[8]; // car  joint5 pillar
//	m_outHandData[2] :=m_handData[3]*256 + m_handData[4]; //car joint7 beamStretch
//	m_outHandData[3] :=m_handData[1]*256 + m_handData[2]; // car joint6  beamRot
//	m_outHandData[4] :=m_handData[5]*256 + m_handData[6]; // joint8 overhang 
//	m_outHandData[5] :=m_handData[9]*256 + m_handData[10];
//	m_outHandData[6] :=m_handData[11]*256 + m_handData[12];
//	m_outHandData[7] :=m_handData[13]*256 + m_handData[14];
//	m_outHandData[8] :=m_handData[15]*256 + m_handData[16];
//END_IF
m_handData := i_joystickDataFromUI;

joystickSignalAnalysis[1]:=LIMIT(0, UDINT_TO_LREAL( m_handData[1]), 1000);
joystickSignalAnalysis[2]:=LIMIT(0, UDINT_TO_LREAL( m_handData[2]), 1000);
joystickSignalAnalysis[3]:=LIMIT(0, UDINT_TO_LREAL( m_handData[3]), 1000);
joystickSignalAnalysis[4]:=LIMIT(0, UDINT_TO_LREAL( m_handData[4]), 1000);
END_METHOD

METHOD ProcessingUIData : BOOL
VAR_IN_OUT CONSTANT
	//UI information, import from UI controller
	i_UIData :ST_CartUIData;
END_VAR
VAR
	i : INT;
END_VAR
m_joystickSignal := joystickSignalAnalysis(m_joystickSignalIO);

m_ctrlEnable:=i_UIData.m_ctrlEnableFromUI;

m_cartDataFromUI.m_standColumnHightLimit := i_UIData.m_standColumnHightLimit;

m_cartDataFromUI.m_cartSpecificPosDraping := GVL_CartControlParameters.g_surgicalDrapingPos;

FOR i := 1 TO g_sArmNum BY 1 DO
	IF i_UIData.m_surgicalSite > 0 AND i_UIData.m_surgicalLocation > 0 THEN
		m_cartDataFromUI.m_cartSpecificPosDocking[i + 4] := GVL_CartControlParameters.g_surgicalOrientPos[i_UIData.m_surgicalSite, i_UIData.m_surgicalLocation,i];
	END_IF
END_FOR

m_surgicalStatusF(CLK:= GVL_interactUI.g_surgicalStatus , Q=> );
IF m_surgicalStatusF.Q THEN
	cartDrapingState := 0;
END_IF

IF NOT (m_cartDataFromUI.m_surgicalSite = i_UIData.m_surgicalSite) OR NOT (m_cartDataFromUI.m_surgicalLocation = i_UIData.m_surgicalLocation) THEN
	cartDockingState := 0;
END_IF

m_cartDataFromUI.m_surgicalSite := i_UIData.m_surgicalSite;
m_cartDataFromUI.m_surgicalLocation := i_UIData.m_surgicalLocation;
END_METHOD

PROPERTY status : ST_CartStatus
GET
status := m_cartStatus;
END_GET
END_PROPERTY

